//     PlcTask Outputs/GVL_iXlinker.EtherCAT_Master_BKCUCX.TcTerminals210_EK1100_2.TcTerminals210_2BK1250.A_0027_KL_6904_Safety_Logic_7_TwinSAFE_Connections.Channel_1.Safety_IB_3 <-> Channel 1/Safety IB 3
//     PlcTask Outputs/GVL_iXlinker.EtherCAT_Master_BKCUCX.TcTerminals210_EK1100_2.TcTerminals210_2BK1250.A_0027_KL_6904_Safety_Logic_7_TwinSAFE_Connections.Channel_1.Safety_IB_4 <-> Channel 1/Safety IB 4
//     PlcTask Outputs/GVL_iXlinker.EtherCAT_Master_BKCUCX.TcTerminals210_EK1100_2.TcTerminals210_2BK1250.A_0027_KL_6904_Safety_Logic_7_TwinSAFE_Connections.Channel_1.Safety_IB_5 <-> Channel 1/Safety IB 5
//     PlcTask Outputs/GVL_iXlinker.EtherCAT_Master_BKCUCX.TcTerminals210_EK1100_2.TcTerminals210_2BK1250.A_0027_KL_6904_Safety_Logic_7_TwinSAFE_Connections.Channel_1.Safety_IB_6 <-> Channel 1/Safety IB 6
//     PlcTask Outputs/GVL_iXlinker.EtherCAT_Master_BKCUCX.TcTerminals210_EK1100_2.TcTerminals210_2BK1250.A_0027_KL_6904_Safety_Logic_7_TwinSAFE_Connections.Channel_1.Safety_IB_7 <-> Channel 1/Safety IB 7
//   PLC/PLC Instance <-> EtherCAT Master BKCUCX/TcTerminals210_EK1100_2/TcTerminals210_2BK1250/A_0028(KL 6904, Safety Logic (15 TwinSAFE Connections))
//     PlcTask Inputs/GVL_iXlinker.EtherCAT_Master_BKCUCX.TcTerminals210_EK1100_2.TcTerminals210_2BK1250.A_0028_KL_6904_Safety_Logic_15_TwinSAFE_Connections.Channel_1.Status <-> Channel 1/Status
//     PlcTask Inputs/GVL_iXlinker.EtherCAT_Master_BKCUCX.TcTerminals210_EK1100_2.TcTerminals210_2BK1250.A_0028_KL_6904_Safety_Logic_15_TwinSAFE_Connections.Channel_1.Register_In <-> Channel 1/Register In
//     PlcTask Inputs/GVL_iXlinker.EtherCAT_Master_BKCUCX.TcTerminals210_EK1100_2.TcTerminals210_2BK1250.A_0028_KL_6904_Safety_Logic_15_TwinSAFE_Connections.Channel_1.Standard_QX_1 <-> Channel 1/Standard QX 1
//     PlcTask Inputs/GVL_iXlinker.EtherCAT_Master_BKCUCX.TcTerminals210_EK1100_2.TcTerminals210_2BK1250.A_0028_KL_6904_Safety_Logic_15_TwinSAFE_Connections.Channel_1.Standard_QX_2 <-> Channel 1/Standard QX 2
//     PlcTask Inputs/GVL_iXlinker.EtherCAT_Master_BKCUCX.TcTerminals210_EK1100_2.TcTerminals210_2BK1250.A_0028_KL_6904_Safety_Logic_15_TwinSAFE_Connections.Channel_1.Standard_QX_3 <-> Channel 1/Standard QX 3
//     PlcTask Inputs/GVL_iXlinker.EtherCAT_Master_BKCUCX.TcTerminals210_EK1100_2.TcTerminals210_2BK1250.A_0028_KL_6904_Safety_Logic_15_TwinSAFE_Connections.Channel_1.Safety_QB_1 <-> Channel 1/Safety QB 1
//     PlcTask Inputs/GVL_iXlinker.EtherCAT_Master_BKCUCX.TcTerminals210_EK1100_2.TcTerminals210_2BK1250.A_0028_KL_6904_Safety_Logic_15_TwinSAFE_Connections.Channel_1.Safety_QB_2 <-> Channel 1/Safety QB 2
//     PlcTask Inputs/GVL_iXlinker.EtherCAT_Master_BKCUCX.TcTerminals210_EK1100_2.TcTerminals210_2BK1250.A_0028_KL_6904_Safety_Logic_15_TwinSAFE_Connections.Channel_1.Safety_QB_3 <-> Channel 1/Safety QB 3
//     PlcTask Inputs/GVL_iXlinker.EtherCAT_Master_BKCUCX.TcTerminals210_EK1100_2.TcTerminals210_2BK1250.A_0028_KL_6904_Safety_Logic_15_TwinSAFE_Connections.Channel_1.Safety_QB_4 <-> Channel 1/Safety QB 4
//     PlcTask Inputs/GVL_iXlinker.EtherCAT_Master_BKCUCX.TcTerminals210_EK1100_2.TcTerminals210_2BK1250.A_0028_KL_6904_Safety_Logic_15_TwinSAFE_Connections.Channel_1.Safety_QB_5 <-> Channel 1/Safety QB 5
//     PlcTask Inputs/GVL_iXlinker.EtherCAT_Master_BKCUCX.TcTerminals210_EK1100_2.TcTerminals210_2BK1250.A_0028_KL_6904_Safety_Logic_15_TwinSAFE_Connections.Channel_1.Safety_QB_6 <-> Channel 1/Safety QB 6
//     PlcTask Inputs/GVL_iXlinker.EtherCAT_Master_BKCUCX.TcTerminals210_EK1100_2.TcTerminals210_2BK1250.A_0028_KL_6904_Safety_Logic_15_TwinSAFE_Connections.Channel_1.Safety_QB_7 <-> Channel 1/Safety QB 7
//     PlcTask Inputs/GVL_iXlinker.EtherCAT_Master_BKCUCX.TcTerminals210_EK1100_2.TcTerminals210_2BK1250.A_0028_KL_6904_Safety_Logic_15_TwinSAFE_Connections.Channel_1.Safety_QB_8 <-> Channel 1/Safety QB 8
//     PlcTask Inputs/GVL_iXlinker.EtherCAT_Master_BKCUCX.TcTerminals210_EK1100_2.TcTerminals210_2BK1250.A_0028_KL_6904_Safety_Logic_15_TwinSAFE_Connections.Channel_1.Safety_QB_9 <-> Channel 1/Safety QB 9
//     PlcTask Inputs/GVL_iXlinker.EtherCAT_Master_BKCUCX.TcTerminals210_EK1100_2.TcTerminals210_2BK1250.A_0028_KL_6904_Safety_Logic_15_TwinSAFE_Connections.Channel_1.Safety_QB_10 <-> Channel 1/Safety QB 10
//     PlcTask Inputs/GVL_iXlinker.EtherCAT_Master_BKCUCX.TcTerminals210_EK1100_2.TcTerminals210_2BK1250.A_0028_KL_6904_Safety_Logic_15_TwinSAFE_Connections.Channel_1.Safety_QB_11 <-> Channel 1/Safety QB 11
//     PlcTask Inputs/GVL_iXlinker.EtherCAT_Master_BKCUCX.TcTerminals210_EK1100_2.TcTerminals210_2BK1250.A_0028_KL_6904_Safety_Logic_15_TwinSAFE_Connections.Channel_1.Safety_QB_12 <-> Channel 1/Safety QB 12
//     PlcTask Inputs/GVL_iXlinker.EtherCAT_Master_BKCUCX.TcTerminals210_EK1100_2.TcTerminals210_2BK1250.A_0028_KL_6904_Safety_Logic_15_TwinSAFE_Connections.Channel_1.Safety_QB_13 <-> Channel 1/Safety QB 13
//     PlcTask Inputs/GVL_iXlinker.EtherCAT_Master_BKCUCX.TcTerminals210_EK1100_2.TcTerminals210_2BK1250.A_0028_KL_6904_Safety_Logic_15_TwinSAFE_Connections.Channel_1.Safety_QB_14 <-> Channel 1/Safety QB 14
//     PlcTask Inputs/GVL_iXlinker.EtherCAT_Master_BKCUCX.TcTerminals210_EK1100_2.TcTerminals210_2BK1250.A_0028_KL_6904_Safety_Logic_15_TwinSAFE_Connections.Channel_1.Safety_QB_15 <-> Channel 1/Safety QB 15
//     PlcTask Outputs/GVL_iXlinker.EtherCAT_Master_BKCUCX.TcTerminals210_EK1100_2.TcTerminals210_2BK1250.A_0028_KL_6904_Safety_Logic_15_TwinSAFE_Connections.Channel_1.Control <-> Channel 1/Control
//     PlcTask Outputs/GVL_iXlinker.EtherCAT_Master_BKCUCX.TcTerminals210_EK1100_2.TcTerminals210_2BK1250.A_0028_KL_6904_Safety_Logic_15_TwinSAFE_Connections.Channel_1.Register_Out <-> Channel 1/Register Out
//     PlcTask Outputs/GVL_iXlinker.EtherCAT_Master_BKCUCX.TcTerminals210_EK1100_2.TcTerminals210_2BK1250.A_0028_KL_6904_Safety_Logic_15_TwinSAFE_Connections.Channel_1.Standard_IX_1 <-> Channel 1/Standard IX 1
//     PlcTask Outputs/GVL_iXlinker.EtherCAT_Master_BKCUCX.TcTerminals210_EK1100_2.TcTerminals210_2BK1250.A_0028_KL_6904_Safety_Logic_15_TwinSAFE_Connections.Channel_1.Standard_IX_2 <-> Channel 1/Standard IX 2
//     PlcTask Outputs/GVL_iXlinker.EtherCAT_Master_BKCUCX.TcTerminals210_EK1100_2.TcTerminals210_2BK1250.A_0028_KL_6904_Safety_Logic_15_TwinSAFE_Connections.Channel_1.Standard_IX_3 <-> Channel 1/Standard IX 3
//     PlcTask Outputs/GVL_iXlinker.EtherCAT_Master_BKCUCX.TcTerminals210_EK1100_2.TcTerminals210_2BK1250.A_0028_KL_6904_Safety_Logic_15_TwinSAFE_Connections.Channel_1.Safety_IB_1 <-> Channel 1/Safety IB 1
//     PlcTask Outputs/GVL_iXlinker.EtherCAT_Master_BKCUCX.TcTerminals210_EK1100_2.TcTerminals210_2BK1250.A_0028_KL_6904_Safety_Logic_15_TwinSAFE_Connections.Channel_1.Safety_IB_2 <-> Channel 1/Safety IB 2
//     PlcTask Outputs/GVL_iXlinker.EtherCAT_Master_BKCUCX.TcTerminals210_EK1100_2.TcTerminals210_2BK1250.A_0028_KL_6904_Safety_Logic_15_TwinSAFE_Connections.Channel_1.Safety_IB_3 <-> Channel 1/Safety IB 3
//     PlcTask Outputs/GVL_iXlinker.EtherCAT_Master_BKCUCX.TcTerminals210_EK1100_2.TcTerminals210_2BK1250.A_0028_KL_6904_Safety_Logic_15_TwinSAFE_Connections.Channel_1.Safety_IB_4 <-> Channel 1/Safety IB 4
//     PlcTask Outputs/GVL_iXlinker.EtherCAT_Master_BKCUCX.TcTerminals210_EK1100_2.TcTerminals210_2BK1250.A_0028_KL_6904_Safety_Logic_15_TwinSAFE_Connections.Channel_1.Safety_IB_5 <-> Channel 1/Safety IB 5
//     PlcTask Outputs/GVL_iXlinker.EtherCAT_Master_BKCUCX.TcTerminals210_EK1100_2.TcTerminals210_2BK1250.A_0028_KL_6904_Safety_Logic_15_TwinSAFE_Connections.Channel_1.Safety_IB_6 <-> Channel 1/Safety IB 6
//     PlcTask Outputs/GVL_iXlinker.EtherCAT_Master_BKCUCX.TcTerminals210_EK1100_2.TcTerminals210_2BK1250.A_0028_KL_6904_Safety_Logic_15_TwinSAFE_Connections.Channel_1.Safety_IB_7 <-> Channel 1/Safety IB 7
//     PlcTask Outputs/GVL_iXlinker.EtherCAT_Master_BKCUCX.TcTerminals210_EK1100_2.TcTerminals210_2BK1250.A_0028_KL_6904_Safety_Logic_15_TwinSAFE_Connections.Channel_1.Safety_IB_8 <-> Channel 1/Safety IB 8
//     PlcTask Outputs/GVL_iXlinker.EtherCAT_Master_BKCUCX.TcTerminals210_EK1100_2.TcTerminals210_2BK1250.A_0028_KL_6904_Safety_Logic_15_TwinSAFE_Connections.Channel_1.Safety_IB_9 <-> Channel 1/Safety IB 9
//     PlcTask Outputs/GVL_iXlinker.EtherCAT_Master_BKCUCX.TcTerminals210_EK1100_2.TcTerminals210_2BK1250.A_0028_KL_6904_Safety_Logic_15_TwinSAFE_Connections.Channel_1.Safety_IB_10 <-> Channel 1/Safety IB 10
//     PlcTask Outputs/GVL_iXlinker.EtherCAT_Master_BKCUCX.TcTerminals210_EK1100_2.TcTerminals210_2BK1250.A_0028_KL_6904_Safety_Logic_15_TwinSAFE_Connections.Channel_1.Safety_IB_11 <-> Channel 1/Safety IB 11
//     PlcTask Outputs/GVL_iXlinker.EtherCAT_Master_BKCUCX.TcTerminals210_EK1100_2.TcTerminals210_2BK1250.A_0028_KL_6904_Safety_Logic_15_TwinSAFE_Connections.Channel_1.Safety_IB_12 <-> Channel 1/Safety IB 12
//     PlcTask Outputs/GVL_iXlinker.EtherCAT_Master_BKCUCX.TcTerminals210_EK1100_2.TcTerminals210_2BK1250.A_0028_KL_6904_Safety_Logic_15_TwinSAFE_Connections.Channel_1.Safety_IB_13 <-> Channel 1/Safety IB 13
//     PlcTask Outputs/GVL_iXlinker.EtherCAT_Master_BKCUCX.TcTerminals210_EK1100_2.TcTerminals210_2BK1250.A_0028_KL_6904_Safety_Logic_15_TwinSAFE_Connections.Channel_1.Safety_IB_14 <-> Channel 1/Safety IB 14
//     PlcTask Outputs/GVL_iXlinker.EtherCAT_Master_BKCUCX.TcTerminals210_EK1100_2.TcTerminals210_2BK1250.A_0028_KL_6904_Safety_Logic_15_TwinSAFE_Connections.Channel_1.Safety_IB_15 <-> Channel 1/Safety IB 15
//   PLC/PLC Instance <-> EtherCAT Master BKCUCX/TcTerminals210_EK1100_2/TcTerminals210_2BK1250/A_0029(KL 8001, Powerterminal (1Ch.))
//     PlcTask Inputs/GVL_iXlinker.EtherCAT_Master_BKCUCX.TcTerminals210_EK1100_2.TcTerminals210_2BK1250.A_0029_KL_8001_Powerterminal_1Ch.Channel_1.State_0 <-> Channel 1/State 0
//     PlcTask Inputs/GVL_iXlinker.EtherCAT_Master_BKCUCX.TcTerminals210_EK1100_2.TcTerminals210_2BK1250.A_0029_KL_8001_Powerterminal_1Ch.Channel_1.Data_In_0 <-> Channel 1/Data In 0
//     PlcTask Inputs/GVL_iXlinker.EtherCAT_Master_BKCUCX.TcTerminals210_EK1100_2.TcTerminals210_2BK1250.A_0029_KL_8001_Powerterminal_1Ch.Channel_1.State_Ext <-> Channel 1/State Ext.
//     PlcTask Outputs/GVL_iXlinker.EtherCAT_Master_BKCUCX.TcTerminals210_EK1100_2.TcTerminals210_2BK1250.A_0029_KL_8001_Powerterminal_1Ch.Channel_1.Ctrl_0 <-> Channel 1/Ctrl 0
//     PlcTask Outputs/GVL_iXlinker.EtherCAT_Master_BKCUCX.TcTerminals210_EK1100_2.TcTerminals210_2BK1250.A_0029_KL_8001_Powerterminal_1Ch.Channel_1.Data_Out_0 <-> Channel 1/Data Out 0
//     PlcTask Outputs/GVL_iXlinker.EtherCAT_Master_BKCUCX.TcTerminals210_EK1100_2.TcTerminals210_2BK1250.A_0029_KL_8001_Powerterminal_1Ch.Channel_1.Ctrl_Ext <-> Channel 1/Ctrl Ext.
//   PLC/PLC Instance <-> EtherCAT Master BKCUCX/TcTerminals210_EK1100_2/TcTerminals210_2BK1250/A_0030(KL 8001, Powerterminal (3 Ch.))
//     PlcTask Inputs/GVL_iXlinker.EtherCAT_Master_BKCUCX.TcTerminals210_EK1100_2.TcTerminals210_2BK1250.A_0030_KL_8001_Powerterminal_3_Ch.Channel_1.State_0 <-> Channel 1/State 0
//     PlcTask Inputs/GVL_iXlinker.EtherCAT_Master_BKCUCX.TcTerminals210_EK1100_2.TcTerminals210_2BK1250.A_0030_KL_8001_Powerterminal_3_Ch.Channel_1.State_1 <-> Channel 1/State 1
//     PlcTask Inputs/GVL_iXlinker.EtherCAT_Master_BKCUCX.TcTerminals210_EK1100_2.TcTerminals210_2BK1250.A_0030_KL_8001_Powerterminal_3_Ch.Channel_1.State_2 <-> Channel 1/State 2
//     PlcTask Inputs/GVL_iXlinker.EtherCAT_Master_BKCUCX.TcTerminals210_EK1100_2.TcTerminals210_2BK1250.A_0030_KL_8001_Powerterminal_3_Ch.Channel_1.Data_In_0 <-> Channel 1/Data In 0
//     PlcTask Inputs/GVL_iXlinker.EtherCAT_Master_BKCUCX.TcTerminals210_EK1100_2.TcTerminals210_2BK1250.A_0030_KL_8001_Powerterminal_3_Ch.Channel_1.Data_In_1 <-> Channel 1/Data In 1
//     PlcTask Inputs/GVL_iXlinker.EtherCAT_Master_BKCUCX.TcTerminals210_EK1100_2.TcTerminals210_2BK1250.A_0030_KL_8001_Powerterminal_3_Ch.Channel_1.Data_In_2 <-> Channel 1/Data In 2
//     PlcTask Inputs/GVL_iXlinker.EtherCAT_Master_BKCUCX.TcTerminals210_EK1100_2.TcTerminals210_2BK1250.A_0030_KL_8001_Powerterminal_3_Ch.Channel_1.State_Ext <-> Channel 1/State Ext.
//     PlcTask Outputs/GVL_iXlinker.EtherCAT_Master_BKCUCX.TcTerminals210_EK1100_2.TcTerminals210_2BK1250.A_0030_KL_8001_Powerterminal_3_Ch.Channel_1.Ctrl_0 <-> Channel 1/Ctrl 0
//     PlcTask Outputs/GVL_iXlinker.EtherCAT_Master_BKCUCX.TcTerminals210_EK1100_2.TcTerminals210_2BK1250.A_0030_KL_8001_Powerterminal_3_Ch.Channel_1.Ctrl_1 <-> Channel 1/Ctrl 1
//     PlcTask Outputs/GVL_iXlinker.EtherCAT_Master_BKCUCX.TcTerminals210_EK1100_2.TcTerminals210_2BK1250.A_0030_KL_8001_Powerterminal_3_Ch.Channel_1.Ctrl_2 <-> Channel 1/Ctrl 2
//     PlcTask Outputs/GVL_iXlinker.EtherCAT_Master_BKCUCX.TcTerminals210_EK1100_2.TcTerminals210_2BK1250.A_0030_KL_8001_Powerterminal_3_Ch.Channel_1.Data_Out_0 <-> Channel 1/Data Out 0
//     PlcTask Outputs/GVL_iXlinker.EtherCAT_Master_BKCUCX.TcTerminals210_EK1100_2.TcTerminals210_2BK1250.A_0030_KL_8001_Powerterminal_3_Ch.Channel_1.Data_Out_1 <-> Channel 1/Data Out 1
//     PlcTask Outputs/GVL_iXlinker.EtherCAT_Master_BKCUCX.TcTerminals210_EK1100_2.TcTerminals210_2BK1250.A_0030_KL_8001_Powerterminal_3_Ch.Channel_1.Data_Out_2 <-> Channel 1/Data Out 2
//     PlcTask Outputs/GVL_iXlinker.EtherCAT_Master_BKCUCX.TcTerminals210_EK1100_2.TcTerminals210_2BK1250.A_0030_KL_8001_Powerterminal_3_Ch.Channel_1.Ctrl_Ext <-> Channel 1/Ctrl Ext.
//   PLC/PLC Instance <-> EtherCAT Master BKCUCX/TcTerminals210_EK1100_2/TcTerminals210_2BK1250/A_0031(KL 8519, 16 digital Input)
//     PlcTask Inputs/GVL_iXlinker.EtherCAT_Master_BKCUCX.TcTerminals210_EK1100_2.TcTerminals210_2BK1250.A_0031_KL_8519_16_digital_Input.Channel_1.State <-> Channel 1/State
//     PlcTask Inputs/GVL_iXlinker.EtherCAT_Master_BKCUCX.TcTerminals210_EK1100_2.TcTerminals210_2BK1250.A_0031_KL_8519_16_digital_Input.Channel_1.Data_In_1 <-> Channel 1/Data In 1
//     PlcTask Inputs/GVL_iXlinker.EtherCAT_Master_BKCUCX.TcTerminals210_EK1100_2.TcTerminals210_2BK1250.A_0031_KL_8519_16_digital_Input.Channel_1.Data_In_2 <-> Channel 1/Data In 2
//     PlcTask Outputs/GVL_iXlinker.EtherCAT_Master_BKCUCX.TcTerminals210_EK1100_2.TcTerminals210_2BK1250.A_0031_KL_8519_16_digital_Input.Channel_1.Ctrl <-> Channel 1/Ctrl
//     PlcTask Outputs/GVL_iXlinker.EtherCAT_Master_BKCUCX.TcTerminals210_EK1100_2.TcTerminals210_2BK1250.A_0031_KL_8519_16_digital_Input.Channel_1.LED_Out_green_1 <-> Channel 1/LED Out green 1
//     PlcTask Outputs/GVL_iXlinker.EtherCAT_Master_BKCUCX.TcTerminals210_EK1100_2.TcTerminals210_2BK1250.A_0031_KL_8519_16_digital_Input.Channel_1.LED_Out_green_2 <-> Channel 1/LED Out green 2
//     PlcTask Outputs/GVL_iXlinker.EtherCAT_Master_BKCUCX.TcTerminals210_EK1100_2.TcTerminals210_2BK1250.A_0031_KL_8519_16_digital_Input.Channel_1.LED_Out_red_1 <-> Channel 1/LED Out red 1
//     PlcTask Outputs/GVL_iXlinker.EtherCAT_Master_BKCUCX.TcTerminals210_EK1100_2.TcTerminals210_2BK1250.A_0031_KL_8519_16_digital_Input.Channel_1.LED_Out_red_2 <-> Channel 1/LED Out red 2
//   PLC/PLC Instance <-> EtherCAT Master BKCUCX/TcTerminals210_EK1100_2/TcTerminals210_2BK1250/A_0032(KL 8524, 2x4 digital Output)
//     PlcTask Inputs/GVL_iXlinker.EtherCAT_Master_BKCUCX.TcTerminals210_EK1100_2.TcTerminals210_2BK1250.A_0032_KL_8524_2x4_digital_Output.Channel_1.State <-> Channel 1/State
//     PlcTask Inputs/GVL_iXlinker.EtherCAT_Master_BKCUCX.TcTerminals210_EK1100_2.TcTerminals210_2BK1250.A_0032_KL_8524_2x4_digital_Output.Channel_1.Auto_Manual_Channel <-> Channel 1/Auto/Manual Channel
//     PlcTask Inputs/GVL_iXlinker.EtherCAT_Master_BKCUCX.TcTerminals210_EK1100_2.TcTerminals210_2BK1250.A_0032_KL_8524_2x4_digital_Output.Channel_1.Switch_mode <-> Channel 1/Switch mode
//     PlcTask Inputs/GVL_iXlinker.EtherCAT_Master_BKCUCX.TcTerminals210_EK1100_2.TcTerminals210_2BK1250.A_0032_KL_8524_2x4_digital_Output.Channel_1.On_Off_Channel <-> Channel 1/On/Off Channel
//     PlcTask Outputs/GVL_iXlinker.EtherCAT_Master_BKCUCX.TcTerminals210_EK1100_2.TcTerminals210_2BK1250.A_0032_KL_8524_2x4_digital_Output.Channel_1.Ctrl <-> Channel 1/Ctrl
//     PlcTask Outputs/GVL_iXlinker.EtherCAT_Master_BKCUCX.TcTerminals210_EK1100_2.TcTerminals210_2BK1250.A_0032_KL_8524_2x4_digital_Output.Channel_1.Switch_mode_Out <-> Channel 1/Switch mode Out
//     PlcTask Outputs/GVL_iXlinker.EtherCAT_Master_BKCUCX.TcTerminals210_EK1100_2.TcTerminals210_2BK1250.A_0032_KL_8524_2x4_digital_Output.Channel_1.Data_Reg_Com <-> Channel 1/Data (Reg.Com)
//     PlcTask Outputs/GVL_iXlinker.EtherCAT_Master_BKCUCX.TcTerminals210_EK1100_2.TcTerminals210_2BK1250.A_0032_KL_8524_2x4_digital_Output.Channel_1.LED_Out_green <-> Channel 1/LED Out green
//     PlcTask Outputs/GVL_iXlinker.EtherCAT_Master_BKCUCX.TcTerminals210_EK1100_2.TcTerminals210_2BK1250.A_0032_KL_8524_2x4_digital_Output.Channel_1.LED_Out_yellow <-> Channel 1/LED Out yellow
//   PLC/PLC Instance <-> EtherCAT Master BKCUCX/TcTerminals210_EK1100_2/TcTerminals210_2BK1250/A_0033(KL 8528, 8 digital Output)
//     PlcTask Inputs/GVL_iXlinker.EtherCAT_Master_BKCUCX.TcTerminals210_EK1100_2.TcTerminals210_2BK1250.A_0033_KL_8528_8_digital_Output.Channel_1.State <-> Channel 1/State
//     PlcTask Inputs/GVL_iXlinker.EtherCAT_Master_BKCUCX.TcTerminals210_EK1100_2.TcTerminals210_2BK1250.A_0033_KL_8528_8_digital_Output.Channel_1.Auto_Manual_Channel <-> Channel 1/Auto/Manual Channel
//     PlcTask Inputs/GVL_iXlinker.EtherCAT_Master_BKCUCX.TcTerminals210_EK1100_2.TcTerminals210_2BK1250.A_0033_KL_8528_8_digital_Output.Channel_1.On_Off_Channel <-> Channel 1/On/Off Channel
//     PlcTask Outputs/GVL_iXlinker.EtherCAT_Master_BKCUCX.TcTerminals210_EK1100_2.TcTerminals210_2BK1250.A_0033_KL_8528_8_digital_Output.Channel_1.Ctrl <-> Channel 1/Ctrl
//     PlcTask Outputs/GVL_iXlinker.EtherCAT_Master_BKCUCX.TcTerminals210_EK1100_2.TcTerminals210_2BK1250.A_0033_KL_8528_8_digital_Output.Channel_1.Out <-> Channel 1/Out
//     PlcTask Outputs/GVL_iXlinker.EtherCAT_Master_BKCUCX.TcTerminals210_EK1100_2.TcTerminals210_2BK1250.A_0033_KL_8528_8_digital_Output.Channel_1.Data_Reg_Com <-> Channel 1/Data (Reg.Com)
//     PlcTask Outputs/GVL_iXlinker.EtherCAT_Master_BKCUCX.TcTerminals210_EK1100_2.TcTerminals210_2BK1250.A_0033_KL_8528_8_digital_Output.Channel_1.LED_Out_green <-> Channel 1/LED Out green
//     PlcTask Outputs/GVL_iXlinker.EtherCAT_Master_BKCUCX.TcTerminals210_EK1100_2.TcTerminals210_2BK1250.A_0033_KL_8528_8_digital_Output.Channel_1.LED_Out_yellow <-> Channel 1/LED Out yellow
//   PLC/PLC Instance <-> EtherCAT Master BKCUCX/TcTerminals210_EK1100_2/TcTerminals210_2BK1250/A_0034(KL 8548, 8 Ch. ana. Output (0..10V))
//     PlcTask Inputs/GVL_iXlinker.EtherCAT_Master_BKCUCX.TcTerminals210_EK1100_2.TcTerminals210_2BK1250.A_0034_KL_8548_8_Ch_ana_Output_0_10V.Channel_1.State <-> Channel 1/State
//     PlcTask Inputs/GVL_iXlinker.EtherCAT_Master_BKCUCX.TcTerminals210_EK1100_2.TcTerminals210_2BK1250.A_0034_KL_8548_8_Ch_ana_Output_0_10V.Channel_2.State <-> Channel 2/State
//     PlcTask Inputs/GVL_iXlinker.EtherCAT_Master_BKCUCX.TcTerminals210_EK1100_2.TcTerminals210_2BK1250.A_0034_KL_8548_8_Ch_ana_Output_0_10V.Channel_3.State <-> Channel 3/State
//     PlcTask Inputs/GVL_iXlinker.EtherCAT_Master_BKCUCX.TcTerminals210_EK1100_2.TcTerminals210_2BK1250.A_0034_KL_8548_8_Ch_ana_Output_0_10V.Channel_4.State <-> Channel 4/State
//     PlcTask Inputs/GVL_iXlinker.EtherCAT_Master_BKCUCX.TcTerminals210_EK1100_2.TcTerminals210_2BK1250.A_0034_KL_8548_8_Ch_ana_Output_0_10V.Channel_5.State <-> Channel 5/State
//     PlcTask Inputs/GVL_iXlinker.EtherCAT_Master_BKCUCX.TcTerminals210_EK1100_2.TcTerminals210_2BK1250.A_0034_KL_8548_8_Ch_ana_Output_0_10V.Channel_6.State <-> Channel 6/State
//     PlcTask Inputs/GVL_iXlinker.EtherCAT_Master_BKCUCX.TcTerminals210_EK1100_2.TcTerminals210_2BK1250.A_0034_KL_8548_8_Ch_ana_Output_0_10V.Channel_7.State <-> Channel 7/State
//     PlcTask Inputs/GVL_iXlinker.EtherCAT_Master_BKCUCX.TcTerminals210_EK1100_2.TcTerminals210_2BK1250.A_0034_KL_8548_8_Ch_ana_Output_0_10V.Channel_8.State <-> Channel 8/State
//     PlcTask Inputs/GVL_iXlinker.EtherCAT_Master_BKCUCX.TcTerminals210_EK1100_2.TcTerminals210_2BK1250.A_0034_KL_8548_8_Ch_ana_Output_0_10V.Channel_1.Data_In <-> Channel 1/Data In
//     PlcTask Inputs/GVL_iXlinker.EtherCAT_Master_BKCUCX.TcTerminals210_EK1100_2.TcTerminals210_2BK1250.A_0034_KL_8548_8_Ch_ana_Output_0_10V.Channel_2.Data_In <-> Channel 2/Data In
//     PlcTask Inputs/GVL_iXlinker.EtherCAT_Master_BKCUCX.TcTerminals210_EK1100_2.TcTerminals210_2BK1250.A_0034_KL_8548_8_Ch_ana_Output_0_10V.Channel_3.Data_In <-> Channel 3/Data In
//     PlcTask Inputs/GVL_iXlinker.EtherCAT_Master_BKCUCX.TcTerminals210_EK1100_2.TcTerminals210_2BK1250.A_0034_KL_8548_8_Ch_ana_Output_0_10V.Channel_4.Data_In <-> Channel 4/Data In
//     PlcTask Inputs/GVL_iXlinker.EtherCAT_Master_BKCUCX.TcTerminals210_EK1100_2.TcTerminals210_2BK1250.A_0034_KL_8548_8_Ch_ana_Output_0_10V.Channel_5.Data_In <-> Channel 5/Data In
//     PlcTask Inputs/GVL_iXlinker.EtherCAT_Master_BKCUCX.TcTerminals210_EK1100_2.TcTerminals210_2BK1250.A_0034_KL_8548_8_Ch_ana_Output_0_10V.Channel_6.Data_In <-> Channel 6/Data In
//     PlcTask Inputs/GVL_iXlinker.EtherCAT_Master_BKCUCX.TcTerminals210_EK1100_2.TcTerminals210_2BK1250.A_0034_KL_8548_8_Ch_ana_Output_0_10V.Channel_7.Data_In <-> Channel 7/Data In
//     PlcTask Inputs/GVL_iXlinker.EtherCAT_Master_BKCUCX.TcTerminals210_EK1100_2.TcTerminals210_2BK1250.A_0034_KL_8548_8_Ch_ana_Output_0_10V.Channel_8.Data_In <-> Channel 8/Data In
//     PlcTask Outputs/GVL_iXlinker.EtherCAT_Master_BKCUCX.TcTerminals210_EK1100_2.TcTerminals210_2BK1250.A_0034_KL_8548_8_Ch_ana_Output_0_10V.Channel_1.Ctrl <-> Channel 1/Ctrl
//     PlcTask Outputs/GVL_iXlinker.EtherCAT_Master_BKCUCX.TcTerminals210_EK1100_2.TcTerminals210_2BK1250.A_0034_KL_8548_8_Ch_ana_Output_0_10V.Channel_2.Ctrl <-> Channel 2/Ctrl
//     PlcTask Outputs/GVL_iXlinker.EtherCAT_Master_BKCUCX.TcTerminals210_EK1100_2.TcTerminals210_2BK1250.A_0034_KL_8548_8_Ch_ana_Output_0_10V.Channel_3.Ctrl <-> Channel 3/Ctrl
//     PlcTask Outputs/GVL_iXlinker.EtherCAT_Master_BKCUCX.TcTerminals210_EK1100_2.TcTerminals210_2BK1250.A_0034_KL_8548_8_Ch_ana_Output_0_10V.Channel_4.Ctrl <-> Channel 4/Ctrl
//     PlcTask Outputs/GVL_iXlinker.EtherCAT_Master_BKCUCX.TcTerminals210_EK1100_2.TcTerminals210_2BK1250.A_0034_KL_8548_8_Ch_ana_Output_0_10V.Channel_5.Ctrl <-> Channel 5/Ctrl
//     PlcTask Outputs/GVL_iXlinker.EtherCAT_Master_BKCUCX.TcTerminals210_EK1100_2.TcTerminals210_2BK1250.A_0034_KL_8548_8_Ch_ana_Output_0_10V.Channel_6.Ctrl <-> Channel 6/Ctrl
//     PlcTask Outputs/GVL_iXlinker.EtherCAT_Master_BKCUCX.TcTerminals210_EK1100_2.TcTerminals210_2BK1250.A_0034_KL_8548_8_Ch_ana_Output_0_10V.Channel_7.Ctrl <-> Channel 7/Ctrl
//     PlcTask Outputs/GVL_iXlinker.EtherCAT_Master_BKCUCX.TcTerminals210_EK1100_2.TcTerminals210_2BK1250.A_0034_KL_8548_8_Ch_ana_Output_0_10V.Channel_8.Ctrl <-> Channel 8/Ctrl
//     PlcTask Outputs/GVL_iXlinker.EtherCAT_Master_BKCUCX.TcTerminals210_EK1100_2.TcTerminals210_2BK1250.A_0034_KL_8548_8_Ch_ana_Output_0_10V.Channel_1.Data_Out <-> Channel 1/Data Out
//     PlcTask Outputs/GVL_iXlinker.EtherCAT_Master_BKCUCX.TcTerminals210_EK1100_2.TcTerminals210_2BK1250.A_0034_KL_8548_8_Ch_ana_Output_0_10V.Channel_2.Data_Out <-> Channel 2/Data Out
//     PlcTask Outputs/GVL_iXlinker.EtherCAT_Master_BKCUCX.TcTerminals210_EK1100_2.TcTerminals210_2BK1250.A_0034_KL_8548_8_Ch_ana_Output_0_10V.Channel_3.Data_Out <-> Channel 3/Data Out
//     PlcTask Outputs/GVL_iXlinker.EtherCAT_Master_BKCUCX.TcTerminals210_EK1100_2.TcTerminals210_2BK1250.A_0034_KL_8548_8_Ch_ana_Output_0_10V.Channel_4.Data_Out <-> Channel 4/Data Out
//     PlcTask Outputs/GVL_iXlinker.EtherCAT_Master_BKCUCX.TcTerminals210_EK1100_2.TcTerminals210_2BK1250.A_0034_KL_8548_8_Ch_ana_Output_0_10V.Channel_5.Data_Out <-> Channel 5/Data Out
//     PlcTask Outputs/GVL_iXlinker.EtherCAT_Master_BKCUCX.TcTerminals210_EK1100_2.TcTerminals210_2BK1250.A_0034_KL_8548_8_Ch_ana_Output_0_10V.Channel_6.Data_Out <-> Channel 6/Data Out
//     PlcTask Outputs/GVL_iXlinker.EtherCAT_Master_BKCUCX.TcTerminals210_EK1100_2.TcTerminals210_2BK1250.A_0034_KL_8548_8_Ch_ana_Output_0_10V.Channel_7.Data_Out <-> Channel 7/Data Out
//     PlcTask Outputs/GVL_iXlinker.EtherCAT_Master_BKCUCX.TcTerminals210_EK1100_2.TcTerminals210_2BK1250.A_0034_KL_8548_8_Ch_ana_Output_0_10V.Channel_8.Data_Out <-> Channel 8/Data Out
//   PLC/PLC Instance <-> EtherCAT Master BKCUCX/TcTerminals210_EK1100_2/TcTerminals210_2BK1250/A_0035(KL 8610, 1 Ch. Adapter KL8601)
//     PlcTask Inputs/GVL_iXlinker.EtherCAT_Master_BKCUCX.TcTerminals210_EK1100_2.TcTerminals210_2BK1250.A_0035_KL_8610_1_Ch_Adapter_KL8601.KL8601_1.State <-> KL8601 - 1/State
//     PlcTask Inputs/GVL_iXlinker.EtherCAT_Master_BKCUCX.TcTerminals210_EK1100_2.TcTerminals210_2BK1250.A_0035_KL_8610_1_Ch_Adapter_KL8601.KL8601_1.Data_In <-> KL8601 - 1/Data In
//     PlcTask Outputs/GVL_iXlinker.EtherCAT_Master_BKCUCX.TcTerminals210_EK1100_2.TcTerminals210_2BK1250.A_0035_KL_8610_1_Ch_Adapter_KL8601.KL8601_1.Ctrl <-> KL8601 - 1/Ctrl
//     PlcTask Outputs/GVL_iXlinker.EtherCAT_Master_BKCUCX.TcTerminals210_EK1100_2.TcTerminals210_2BK1250.A_0035_KL_8610_1_Ch_Adapter_KL8601.KL8601_1.Data_Out <-> KL8601 - 1/Data Out
//   PLC/PLC Instance <-> EtherCAT Master BKCUCX/TcTerminals210_EK1100_2/TcTerminals210_2BK1250/A_0036(KL 8610, 2 Ch. Adapter KL8601)
//     PlcTask Inputs/GVL_iXlinker.EtherCAT_Master_BKCUCX.TcTerminals210_EK1100_2.TcTerminals210_2BK1250.A_0036_KL_8610_2_Ch_Adapter_KL8601.KL8601_1.State <-> KL8601 - 1/State
//     PlcTask Inputs/GVL_iXlinker.EtherCAT_Master_BKCUCX.TcTerminals210_EK1100_2.TcTerminals210_2BK1250.A_0036_KL_8610_2_Ch_Adapter_KL8601.KL8601_2.State <-> KL8601 - 2/State
//     PlcTask Inputs/GVL_iXlinker.EtherCAT_Master_BKCUCX.TcTerminals210_EK1100_2.TcTerminals210_2BK1250.A_0036_KL_8610_2_Ch_Adapter_KL8601.KL8601_1.Data_In <-> KL8601 - 1/Data In
//     PlcTask Inputs/GVL_iXlinker.EtherCAT_Master_BKCUCX.TcTerminals210_EK1100_2.TcTerminals210_2BK1250.A_0036_KL_8610_2_Ch_Adapter_KL8601.KL8601_2.Data_In <-> KL8601 - 2/Data In
//     PlcTask Outputs/GVL_iXlinker.EtherCAT_Master_BKCUCX.TcTerminals210_EK1100_2.TcTerminals210_2BK1250.A_0036_KL_8610_2_Ch_Adapter_KL8601.KL8601_1.Ctrl <-> KL8601 - 1/Ctrl
//     PlcTask Outputs/GVL_iXlinker.EtherCAT_Master_BKCUCX.TcTerminals210_EK1100_2.TcTerminals210_2BK1250.A_0036_KL_8610_2_Ch_Adapter_KL8601.KL8601_2.Ctrl <-> KL8601 - 2/Ctrl
//     PlcTask Outputs/GVL_iXlinker.EtherCAT_Master_BKCUCX.TcTerminals210_EK1100_2.TcTerminals210_2BK1250.A_0036_KL_8610_2_Ch_Adapter_KL8601.KL8601_1.Data_Out <-> KL8601 - 1/Data Out
//     PlcTask Outputs/GVL_iXlinker.EtherCAT_Master_BKCUCX.TcTerminals210_EK1100_2.TcTerminals210_2BK1250.A_0036_KL_8610_2_Ch_Adapter_KL8601.KL8601_2.Data_Out <-> KL8601 - 2/Data Out
//   PLC/PLC Instance <-> EtherCAT Master BKCUCX/TcTerminals210_EK1100_2/TcTerminals210_2BK1250/A_0037(KL 8610, 3 Ch. Adapter KL8601)
//     PlcTask Inputs/GVL_iXlinker.EtherCAT_Master_BKCUCX.TcTerminals210_EK1100_2.TcTerminals210_2BK1250.A_0037_KL_8610_3_Ch_Adapter_KL8601.KL8601_1.State <-> KL8601 - 1/State
//     PlcTask Inputs/GVL_iXlinker.EtherCAT_Master_BKCUCX.TcTerminals210_EK1100_2.TcTerminals210_2BK1250.A_0037_KL_8610_3_Ch_Adapter_KL8601.KL8601_2.State <-> KL8601 - 2/State
//     PlcTask Inputs/GVL_iXlinker.EtherCAT_Master_BKCUCX.TcTerminals210_EK1100_2.TcTerminals210_2BK1250.A_0037_KL_8610_3_Ch_Adapter_KL8601.KL8601_3.State <-> KL8601 - 3/State
//     PlcTask Inputs/GVL_iXlinker.EtherCAT_Master_BKCUCX.TcTerminals210_EK1100_2.TcTerminals210_2BK1250.A_0037_KL_8610_3_Ch_Adapter_KL8601.KL8601_1.Data_In <-> KL8601 - 1/Data In
//     PlcTask Inputs/GVL_iXlinker.EtherCAT_Master_BKCUCX.TcTerminals210_EK1100_2.TcTerminals210_2BK1250.A_0037_KL_8610_3_Ch_Adapter_KL8601.KL8601_2.Data_In <-> KL8601 - 2/Data In
//     PlcTask Inputs/GVL_iXlinker.EtherCAT_Master_BKCUCX.TcTerminals210_EK1100_2.TcTerminals210_2BK1250.A_0037_KL_8610_3_Ch_Adapter_KL8601.KL8601_3.Data_In <-> KL8601 - 3/Data In
//     PlcTask Outputs/GVL_iXlinker.EtherCAT_Master_BKCUCX.TcTerminals210_EK1100_2.TcTerminals210_2BK1250.A_0037_KL_8610_3_Ch_Adapter_KL8601.KL8601_1.Ctrl <-> KL8601 - 1/Ctrl
//     PlcTask Outputs/GVL_iXlinker.EtherCAT_Master_BKCUCX.TcTerminals210_EK1100_2.TcTerminals210_2BK1250.A_0037_KL_8610_3_Ch_Adapter_KL8601.KL8601_2.Ctrl <-> KL8601 - 2/Ctrl
//     PlcTask Outputs/GVL_iXlinker.EtherCAT_Master_BKCUCX.TcTerminals210_EK1100_2.TcTerminals210_2BK1250.A_0037_KL_8610_3_Ch_Adapter_KL8601.KL8601_3.Ctrl <-> KL8601 - 3/Ctrl
//     PlcTask Outputs/GVL_iXlinker.EtherCAT_Master_BKCUCX.TcTerminals210_EK1100_2.TcTerminals210_2BK1250.A_0037_KL_8610_3_Ch_Adapter_KL8601.KL8601_1.Data_Out <-> KL8601 - 1/Data Out
//     PlcTask Outputs/GVL_iXlinker.EtherCAT_Master_BKCUCX.TcTerminals210_EK1100_2.TcTerminals210_2BK1250.A_0037_KL_8610_3_Ch_Adapter_KL8601.KL8601_2.Data_Out <-> KL8601 - 2/Data Out
//     PlcTask Outputs/GVL_iXlinker.EtherCAT_Master_BKCUCX.TcTerminals210_EK1100_2.TcTerminals210_2BK1250.A_0037_KL_8610_3_Ch_Adapter_KL8601.KL8601_3.Data_Out <-> KL8601 - 3/Data Out
//   PLC/PLC Instance <-> EtherCAT Master BKCUCX/TcTerminals210_EK1100_2/TcTerminals210_2BK1250/A_0038(KL 8610, 4 Ch. Adapter KL8601)
//     PlcTask Inputs/GVL_iXlinker.EtherCAT_Master_BKCUCX.TcTerminals210_EK1100_2.TcTerminals210_2BK1250.A_0038_KL_8610_4_Ch_Adapter_KL8601.KL8601_1.State <-> KL8601 - 1/State
//     PlcTask Inputs/GVL_iXlinker.EtherCAT_Master_BKCUCX.TcTerminals210_EK1100_2.TcTerminals210_2BK1250.A_0038_KL_8610_4_Ch_Adapter_KL8601.KL8601_2.State <-> KL8601 - 2/State
//     PlcTask Inputs/GVL_iXlinker.EtherCAT_Master_BKCUCX.TcTerminals210_EK1100_2.TcTerminals210_2BK1250.A_0038_KL_8610_4_Ch_Adapter_KL8601.KL8601_3.State <-> KL8601 - 3/State
//     PlcTask Inputs/GVL_iXlinker.EtherCAT_Master_BKCUCX.TcTerminals210_EK1100_2.TcTerminals210_2BK1250.A_0038_KL_8610_4_Ch_Adapter_KL8601.KL8601_4.State <-> KL8601 - 4/State
//     PlcTask Inputs/GVL_iXlinker.EtherCAT_Master_BKCUCX.TcTerminals210_EK1100_2.TcTerminals210_2BK1250.A_0038_KL_8610_4_Ch_Adapter_KL8601.KL8601_1.Data_In <-> KL8601 - 1/Data In
//     PlcTask Inputs/GVL_iXlinker.EtherCAT_Master_BKCUCX.TcTerminals210_EK1100_2.TcTerminals210_2BK1250.A_0038_KL_8610_4_Ch_Adapter_KL8601.KL8601_2.Data_In <-> KL8601 - 2/Data In
//     PlcTask Inputs/GVL_iXlinker.EtherCAT_Master_BKCUCX.TcTerminals210_EK1100_2.TcTerminals210_2BK1250.A_0038_KL_8610_4_Ch_Adapter_KL8601.KL8601_3.Data_In <-> KL8601 - 3/Data In
//     PlcTask Inputs/GVL_iXlinker.EtherCAT_Master_BKCUCX.TcTerminals210_EK1100_2.TcTerminals210_2BK1250.A_0038_KL_8610_4_Ch_Adapter_KL8601.KL8601_4.Data_In <-> KL8601 - 4/Data In
//     PlcTask Outputs/GVL_iXlinker.EtherCAT_Master_BKCUCX.TcTerminals210_EK1100_2.TcTerminals210_2BK1250.A_0038_KL_8610_4_Ch_Adapter_KL8601.KL8601_1.Ctrl <-> KL8601 - 1/Ctrl
//     PlcTask Outputs/GVL_iXlinker.EtherCAT_Master_BKCUCX.TcTerminals210_EK1100_2.TcTerminals210_2BK1250.A_0038_KL_8610_4_Ch_Adapter_KL8601.KL8601_2.Ctrl <-> KL8601 - 2/Ctrl
//     PlcTask Outputs/GVL_iXlinker.EtherCAT_Master_BKCUCX.TcTerminals210_EK1100_2.TcTerminals210_2BK1250.A_0038_KL_8610_4_Ch_Adapter_KL8601.KL8601_3.Ctrl <-> KL8601 - 3/Ctrl
//     PlcTask Outputs/GVL_iXlinker.EtherCAT_Master_BKCUCX.TcTerminals210_EK1100_2.TcTerminals210_2BK1250.A_0038_KL_8610_4_Ch_Adapter_KL8601.KL8601_4.Ctrl <-> KL8601 - 4/Ctrl
//     PlcTask Outputs/GVL_iXlinker.EtherCAT_Master_BKCUCX.TcTerminals210_EK1100_2.TcTerminals210_2BK1250.A_0038_KL_8610_4_Ch_Adapter_KL8601.KL8601_1.Data_Out <-> KL8601 - 1/Data Out
//     PlcTask Outputs/GVL_iXlinker.EtherCAT_Master_BKCUCX.TcTerminals210_EK1100_2.TcTerminals210_2BK1250.A_0038_KL_8610_4_Ch_Adapter_KL8601.KL8601_2.Data_Out <-> KL8601 - 2/Data Out
//     PlcTask Outputs/GVL_iXlinker.EtherCAT_Master_BKCUCX.TcTerminals210_EK1100_2.TcTerminals210_2BK1250.A_0038_KL_8610_4_Ch_Adapter_KL8601.KL8601_3.Data_Out <-> KL8601 - 3/Data Out
//     PlcTask Outputs/GVL_iXlinker.EtherCAT_Master_BKCUCX.TcTerminals210_EK1100_2.TcTerminals210_2BK1250.A_0038_KL_8610_4_Ch_Adapter_KL8601.KL8601_4.Data_Out <-> KL8601 - 4/Data Out
//   PLC/PLC Instance <-> EtherCAT Master BKCUCX/TcTerminals210_EK1100_2/TcTerminals210_2BK1250/A_0039(KL 8610, 5 Ch. Adapter KL8601)
//     PlcTask Inputs/GVL_iXlinker.EtherCAT_Master_BKCUCX.TcTerminals210_EK1100_2.TcTerminals210_2BK1250.A_0039_KL_8610_5_Ch_Adapter_KL8601.KL8601_1.State <-> KL8601 - 1/State
//     PlcTask Inputs/GVL_iXlinker.EtherCAT_Master_BKCUCX.TcTerminals210_EK1100_2.TcTerminals210_2BK1250.A_0039_KL_8610_5_Ch_Adapter_KL8601.KL8601_2.State <-> KL8601 - 2/State
//     PlcTask Inputs/GVL_iXlinker.EtherCAT_Master_BKCUCX.TcTerminals210_EK1100_2.TcTerminals210_2BK1250.A_0039_KL_8610_5_Ch_Adapter_KL8601.KL8601_3.State <-> KL8601 - 3/State
//     PlcTask Inputs/GVL_iXlinker.EtherCAT_Master_BKCUCX.TcTerminals210_EK1100_2.TcTerminals210_2BK1250.A_0039_KL_8610_5_Ch_Adapter_KL8601.KL8601_4.State <-> KL8601 - 4/State
//     PlcTask Inputs/GVL_iXlinker.EtherCAT_Master_BKCUCX.TcTerminals210_EK1100_2.TcTerminals210_2BK1250.A_0039_KL_8610_5_Ch_Adapter_KL8601.KL8601_5.State <-> KL8601 - 5/State
//     PlcTask Inputs/GVL_iXlinker.EtherCAT_Master_BKCUCX.TcTerminals210_EK1100_2.TcTerminals210_2BK1250.A_0039_KL_8610_5_Ch_Adapter_KL8601.KL8601_1.Data_In <-> KL8601 - 1/Data In
//     PlcTask Inputs/GVL_iXlinker.EtherCAT_Master_BKCUCX.TcTerminals210_EK1100_2.TcTerminals210_2BK1250.A_0039_KL_8610_5_Ch_Adapter_KL8601.KL8601_2.Data_In <-> KL8601 - 2/Data In
//     PlcTask Inputs/GVL_iXlinker.EtherCAT_Master_BKCUCX.TcTerminals210_EK1100_2.TcTerminals210_2BK1250.A_0039_KL_8610_5_Ch_Adapter_KL8601.KL8601_3.Data_In <-> KL8601 - 3/Data In
//     PlcTask Inputs/GVL_iXlinker.EtherCAT_Master_BKCUCX.TcTerminals210_EK1100_2.TcTerminals210_2BK1250.A_0039_KL_8610_5_Ch_Adapter_KL8601.KL8601_4.Data_In <-> KL8601 - 4/Data In
//     PlcTask Inputs/GVL_iXlinker.EtherCAT_Master_BKCUCX.TcTerminals210_EK1100_2.TcTerminals210_2BK1250.A_0039_KL_8610_5_Ch_Adapter_KL8601.KL8601_5.Data_In <-> KL8601 - 5/Data In
//     PlcTask Outputs/GVL_iXlinker.EtherCAT_Master_BKCUCX.TcTerminals210_EK1100_2.TcTerminals210_2BK1250.A_0039_KL_8610_5_Ch_Adapter_KL8601.KL8601_1.Ctrl <-> KL8601 - 1/Ctrl
//     PlcTask Outputs/GVL_iXlinker.EtherCAT_Master_BKCUCX.TcTerminals210_EK1100_2.TcTerminals210_2BK1250.A_0039_KL_8610_5_Ch_Adapter_KL8601.KL8601_2.Ctrl <-> KL8601 - 2/Ctrl
//     PlcTask Outputs/GVL_iXlinker.EtherCAT_Master_BKCUCX.TcTerminals210_EK1100_2.TcTerminals210_2BK1250.A_0039_KL_8610_5_Ch_Adapter_KL8601.KL8601_3.Ctrl <-> KL8601 - 3/Ctrl
//     PlcTask Outputs/GVL_iXlinker.EtherCAT_Master_BKCUCX.TcTerminals210_EK1100_2.TcTerminals210_2BK1250.A_0039_KL_8610_5_Ch_Adapter_KL8601.KL8601_4.Ctrl <-> KL8601 - 4/Ctrl
//     PlcTask Outputs/GVL_iXlinker.EtherCAT_Master_BKCUCX.TcTerminals210_EK1100_2.TcTerminals210_2BK1250.A_0039_KL_8610_5_Ch_Adapter_KL8601.KL8601_5.Ctrl <-> KL8601 - 5/Ctrl
//     PlcTask Outputs/GVL_iXlinker.EtherCAT_Master_BKCUCX.TcTerminals210_EK1100_2.TcTerminals210_2BK1250.A_0039_KL_8610_5_Ch_Adapter_KL8601.KL8601_1.Data_Out <-> KL8601 - 1/Data Out
//     PlcTask Outputs/GVL_iXlinker.EtherCAT_Master_BKCUCX.TcTerminals210_EK1100_2.TcTerminals210_2BK1250.A_0039_KL_8610_5_Ch_Adapter_KL8601.KL8601_2.Data_Out <-> KL8601 - 2/Data Out
//     PlcTask Outputs/GVL_iXlinker.EtherCAT_Master_BKCUCX.TcTerminals210_EK1100_2.TcTerminals210_2BK1250.A_0039_KL_8610_5_Ch_Adapter_KL8601.KL8601_3.Data_Out <-> KL8601 - 3/Data Out
//     PlcTask Outputs/GVL_iXlinker.EtherCAT_Master_BKCUCX.TcTerminals210_EK1100_2.TcTerminals210_2BK1250.A_0039_KL_8610_5_Ch_Adapter_KL8601.KL8601_4.Data_Out <-> KL8601 - 4/Data Out
//     PlcTask Outputs/GVL_iXlinker.EtherCAT_Master_BKCUCX.TcTerminals210_EK1100_2.TcTerminals210_2BK1250.A_0039_KL_8610_5_Ch_Adapter_KL8601.KL8601_5.Data_Out <-> KL8601 - 5/Data Out
//   PLC/PLC Instance <-> EtherCAT Master BKCUCX/TcTerminals210_EK1100_2/TcTerminals210_2BK1250/A_0040(KL 8610, 6 Ch. Adapter KL8601)
//     PlcTask Inputs/GVL_iXlinker.EtherCAT_Master_BKCUCX.TcTerminals210_EK1100_2.TcTerminals210_2BK1250.A_0040_KL_8610_6_Ch_Adapter_KL8601.KL8601_1.State <-> KL8601 - 1/State
//     PlcTask Inputs/GVL_iXlinker.EtherCAT_Master_BKCUCX.TcTerminals210_EK1100_2.TcTerminals210_2BK1250.A_0040_KL_8610_6_Ch_Adapter_KL8601.KL8601_2.State <-> KL8601 - 2/State
//     PlcTask Inputs/GVL_iXlinker.EtherCAT_Master_BKCUCX.TcTerminals210_EK1100_2.TcTerminals210_2BK1250.A_0040_KL_8610_6_Ch_Adapter_KL8601.KL8601_3.State <-> KL8601 - 3/State
//     PlcTask Inputs/GVL_iXlinker.EtherCAT_Master_BKCUCX.TcTerminals210_EK1100_2.TcTerminals210_2BK1250.A_0040_KL_8610_6_Ch_Adapter_KL8601.KL8601_4.State <-> KL8601 - 4/State
//     PlcTask Inputs/GVL_iXlinker.EtherCAT_Master_BKCUCX.TcTerminals210_EK1100_2.TcTerminals210_2BK1250.A_0040_KL_8610_6_Ch_Adapter_KL8601.KL8601_5.State <-> KL8601 - 5/State
//     PlcTask Inputs/GVL_iXlinker.EtherCAT_Master_BKCUCX.TcTerminals210_EK1100_2.TcTerminals210_2BK1250.A_0040_KL_8610_6_Ch_Adapter_KL8601.KL8601_6.State <-> KL8601 - 6/State
//     PlcTask Inputs/GVL_iXlinker.EtherCAT_Master_BKCUCX.TcTerminals210_EK1100_2.TcTerminals210_2BK1250.A_0040_KL_8610_6_Ch_Adapter_KL8601.KL8601_1.Data_In <-> KL8601 - 1/Data In
//     PlcTask Inputs/GVL_iXlinker.EtherCAT_Master_BKCUCX.TcTerminals210_EK1100_2.TcTerminals210_2BK1250.A_0040_KL_8610_6_Ch_Adapter_KL8601.KL8601_2.Data_In <-> KL8601 - 2/Data In
//     PlcTask Inputs/GVL_iXlinker.EtherCAT_Master_BKCUCX.TcTerminals210_EK1100_2.TcTerminals210_2BK1250.A_0040_KL_8610_6_Ch_Adapter_KL8601.KL8601_3.Data_In <-> KL8601 - 3/Data In
//     PlcTask Inputs/GVL_iXlinker.EtherCAT_Master_BKCUCX.TcTerminals210_EK1100_2.TcTerminals210_2BK1250.A_0040_KL_8610_6_Ch_Adapter_KL8601.KL8601_4.Data_In <-> KL8601 - 4/Data In
//     PlcTask Inputs/GVL_iXlinker.EtherCAT_Master_BKCUCX.TcTerminals210_EK1100_2.TcTerminals210_2BK1250.A_0040_KL_8610_6_Ch_Adapter_KL8601.KL8601_5.Data_In <-> KL8601 - 5/Data In
//     PlcTask Inputs/GVL_iXlinker.EtherCAT_Master_BKCUCX.TcTerminals210_EK1100_2.TcTerminals210_2BK1250.A_0040_KL_8610_6_Ch_Adapter_KL8601.KL8601_6.Data_In <-> KL8601 - 6/Data In
//     PlcTask Outputs/GVL_iXlinker.EtherCAT_Master_BKCUCX.TcTerminals210_EK1100_2.TcTerminals210_2BK1250.A_0040_KL_8610_6_Ch_Adapter_KL8601.KL8601_1.Ctrl <-> KL8601 - 1/Ctrl
//     PlcTask Outputs/GVL_iXlinker.EtherCAT_Master_BKCUCX.TcTerminals210_EK1100_2.TcTerminals210_2BK1250.A_0040_KL_8610_6_Ch_Adapter_KL8601.KL8601_2.Ctrl <-> KL8601 - 2/Ctrl
//     PlcTask Outputs/GVL_iXlinker.EtherCAT_Master_BKCUCX.TcTerminals210_EK1100_2.TcTerminals210_2BK1250.A_0040_KL_8610_6_Ch_Adapter_KL8601.KL8601_3.Ctrl <-> KL8601 - 3/Ctrl
//     PlcTask Outputs/GVL_iXlinker.EtherCAT_Master_BKCUCX.TcTerminals210_EK1100_2.TcTerminals210_2BK1250.A_0040_KL_8610_6_Ch_Adapter_KL8601.KL8601_4.Ctrl <-> KL8601 - 4/Ctrl
//     PlcTask Outputs/GVL_iXlinker.EtherCAT_Master_BKCUCX.TcTerminals210_EK1100_2.TcTerminals210_2BK1250.A_0040_KL_8610_6_Ch_Adapter_KL8601.KL8601_5.Ctrl <-> KL8601 - 5/Ctrl
//     PlcTask Outputs/GVL_iXlinker.EtherCAT_Master_BKCUCX.TcTerminals210_EK1100_2.TcTerminals210_2BK1250.A_0040_KL_8610_6_Ch_Adapter_KL8601.KL8601_6.Ctrl <-> KL8601 - 6/Ctrl
//     PlcTask Outputs/GVL_iXlinker.EtherCAT_Master_BKCUCX.TcTerminals210_EK1100_2.TcTerminals210_2BK1250.A_0040_KL_8610_6_Ch_Adapter_KL8601.KL8601_1.Data_Out <-> KL8601 - 1/Data Out
//     PlcTask Outputs/GVL_iXlinker.EtherCAT_Master_BKCUCX.TcTerminals210_EK1100_2.TcTerminals210_2BK1250.A_0040_KL_8610_6_Ch_Adapter_KL8601.KL8601_2.Data_Out <-> KL8601 - 2/Data Out
//     PlcTask Outputs/GVL_iXlinker.EtherCAT_Master_BKCUCX.TcTerminals210_EK1100_2.TcTerminals210_2BK1250.A_0040_KL_8610_6_Ch_Adapter_KL8601.KL8601_3.Data_Out <-> KL8601 - 3/Data Out
//     PlcTask Outputs/GVL_iXlinker.EtherCAT_Master_BKCUCX.TcTerminals210_EK1100_2.TcTerminals210_2BK1250.A_0040_KL_8610_6_Ch_Adapter_KL8601.KL8601_4.Data_Out <-> KL8601 - 4/Data Out
//     PlcTask Outputs/GVL_iXlinker.EtherCAT_Master_BKCUCX.TcTerminals210_EK1100_2.TcTerminals210_2BK1250.A_0040_KL_8610_6_Ch_Adapter_KL8601.KL8601_5.Data_Out <-> KL8601 - 5/Data Out
//     PlcTask Outputs/GVL_iXlinker.EtherCAT_Master_BKCUCX.TcTerminals210_EK1100_2.TcTerminals210_2BK1250.A_0040_KL_8610_6_Ch_Adapter_KL8601.KL8601_6.Data_Out <-> KL8601 - 6/Data Out
//   PLC/PLC Instance <-> EtherCAT Master BKCUCX/TcTerminals210_EK1100_2/TcTerminals210_2BK1250/A_0041(KL 8610, 7 Ch. Adapter KL8601)
//     PlcTask Inputs/GVL_iXlinker.EtherCAT_Master_BKCUCX.TcTerminals210_EK1100_2.TcTerminals210_2BK1250.A_0041_KL_8610_7_Ch_Adapter_KL8601.KL8601_1.State <-> KL8601 - 1/State
//     PlcTask Inputs/GVL_iXlinker.EtherCAT_Master_BKCUCX.TcTerminals210_EK1100_2.TcTerminals210_2BK1250.A_0041_KL_8610_7_Ch_Adapter_KL8601.KL8601_2.State <-> KL8601 - 2/State
//     PlcTask Inputs/GVL_iXlinker.EtherCAT_Master_BKCUCX.TcTerminals210_EK1100_2.TcTerminals210_2BK1250.A_0041_KL_8610_7_Ch_Adapter_KL8601.KL8601_3.State <-> KL8601 - 3/State
//     PlcTask Inputs/GVL_iXlinker.EtherCAT_Master_BKCUCX.TcTerminals210_EK1100_2.TcTerminals210_2BK1250.A_0041_KL_8610_7_Ch_Adapter_KL8601.KL8601_4.State <-> KL8601 - 4/State
//     PlcTask Inputs/GVL_iXlinker.EtherCAT_Master_BKCUCX.TcTerminals210_EK1100_2.TcTerminals210_2BK1250.A_0041_KL_8610_7_Ch_Adapter_KL8601.KL8601_5.State <-> KL8601 - 5/State
//     PlcTask Inputs/GVL_iXlinker.EtherCAT_Master_BKCUCX.TcTerminals210_EK1100_2.TcTerminals210_2BK1250.A_0041_KL_8610_7_Ch_Adapter_KL8601.KL8601_6.State <-> KL8601 - 6/State
//     PlcTask Inputs/GVL_iXlinker.EtherCAT_Master_BKCUCX.TcTerminals210_EK1100_2.TcTerminals210_2BK1250.A_0041_KL_8610_7_Ch_Adapter_KL8601.KL8601_7.State <-> KL8601 - 7/State
//     PlcTask Inputs/GVL_iXlinker.EtherCAT_Master_BKCUCX.TcTerminals210_EK1100_2.TcTerminals210_2BK1250.A_0041_KL_8610_7_Ch_Adapter_KL8601.KL8601_1.Data_In <-> KL8601 - 1/Data In
//     PlcTask Inputs/GVL_iXlinker.EtherCAT_Master_BKCUCX.TcTerminals210_EK1100_2.TcTerminals210_2BK1250.A_0041_KL_8610_7_Ch_Adapter_KL8601.KL8601_2.Data_In <-> KL8601 - 2/Data In
//     PlcTask Inputs/GVL_iXlinker.EtherCAT_Master_BKCUCX.TcTerminals210_EK1100_2.TcTerminals210_2BK1250.A_0041_KL_8610_7_Ch_Adapter_KL8601.KL8601_3.Data_In <-> KL8601 - 3/Data In
//     PlcTask Inputs/GVL_iXlinker.EtherCAT_Master_BKCUCX.TcTerminals210_EK1100_2.TcTerminals210_2BK1250.A_0041_KL_8610_7_Ch_Adapter_KL8601.KL8601_4.Data_In <-> KL8601 - 4/Data In
//     PlcTask Inputs/GVL_iXlinker.EtherCAT_Master_BKCUCX.TcTerminals210_EK1100_2.TcTerminals210_2BK1250.A_0041_KL_8610_7_Ch_Adapter_KL8601.KL8601_5.Data_In <-> KL8601 - 5/Data In
//     PlcTask Inputs/GVL_iXlinker.EtherCAT_Master_BKCUCX.TcTerminals210_EK1100_2.TcTerminals210_2BK1250.A_0041_KL_8610_7_Ch_Adapter_KL8601.KL8601_6.Data_In <-> KL8601 - 6/Data In
//     PlcTask Inputs/GVL_iXlinker.EtherCAT_Master_BKCUCX.TcTerminals210_EK1100_2.TcTerminals210_2BK1250.A_0041_KL_8610_7_Ch_Adapter_KL8601.KL8601_7.Data_In <-> KL8601 - 7/Data In
//     PlcTask Outputs/GVL_iXlinker.EtherCAT_Master_BKCUCX.TcTerminals210_EK1100_2.TcTerminals210_2BK1250.A_0041_KL_8610_7_Ch_Adapter_KL8601.KL8601_1.Ctrl <-> KL8601 - 1/Ctrl
//     PlcTask Outputs/GVL_iXlinker.EtherCAT_Master_BKCUCX.TcTerminals210_EK1100_2.TcTerminals210_2BK1250.A_0041_KL_8610_7_Ch_Adapter_KL8601.KL8601_2.Ctrl <-> KL8601 - 2/Ctrl
//     PlcTask Outputs/GVL_iXlinker.EtherCAT_Master_BKCUCX.TcTerminals210_EK1100_2.TcTerminals210_2BK1250.A_0041_KL_8610_7_Ch_Adapter_KL8601.KL8601_3.Ctrl <-> KL8601 - 3/Ctrl
//     PlcTask Outputs/GVL_iXlinker.EtherCAT_Master_BKCUCX.TcTerminals210_EK1100_2.TcTerminals210_2BK1250.A_0041_KL_8610_7_Ch_Adapter_KL8601.KL8601_4.Ctrl <-> KL8601 - 4/Ctrl
//     PlcTask Outputs/GVL_iXlinker.EtherCAT_Master_BKCUCX.TcTerminals210_EK1100_2.TcTerminals210_2BK1250.A_0041_KL_8610_7_Ch_Adapter_KL8601.KL8601_5.Ctrl <-> KL8601 - 5/Ctrl
//     PlcTask Outputs/GVL_iXlinker.EtherCAT_Master_BKCUCX.TcTerminals210_EK1100_2.TcTerminals210_2BK1250.A_0041_KL_8610_7_Ch_Adapter_KL8601.KL8601_6.Ctrl <-> KL8601 - 6/Ctrl
//     PlcTask Outputs/GVL_iXlinker.EtherCAT_Master_BKCUCX.TcTerminals210_EK1100_2.TcTerminals210_2BK1250.A_0041_KL_8610_7_Ch_Adapter_KL8601.KL8601_7.Ctrl <-> KL8601 - 7/Ctrl
//     PlcTask Outputs/GVL_iXlinker.EtherCAT_Master_BKCUCX.TcTerminals210_EK1100_2.TcTerminals210_2BK1250.A_0041_KL_8610_7_Ch_Adapter_KL8601.KL8601_1.Data_Out <-> KL8601 - 1/Data Out
//     PlcTask Outputs/GVL_iXlinker.EtherCAT_Master_BKCUCX.TcTerminals210_EK1100_2.TcTerminals210_2BK1250.A_0041_KL_8610_7_Ch_Adapter_KL8601.KL8601_2.Data_Out <-> KL8601 - 2/Data Out
//     PlcTask Outputs/GVL_iXlinker.EtherCAT_Master_BKCUCX.TcTerminals210_EK1100_2.TcTerminals210_2BK1250.A_0041_KL_8610_7_Ch_Adapter_KL8601.KL8601_3.Data_Out <-> KL8601 - 3/Data Out
//     PlcTask Outputs/GVL_iXlinker.EtherCAT_Master_BKCUCX.TcTerminals210_EK1100_2.TcTerminals210_2BK1250.A_0041_KL_8610_7_Ch_Adapter_KL8601.KL8601_4.Data_Out <-> KL8601 - 4/Data Out
//     PlcTask Outputs/GVL_iXlinker.EtherCAT_Master_BKCUCX.TcTerminals210_EK1100_2.TcTerminals210_2BK1250.A_0041_KL_8610_7_Ch_Adapter_KL8601.KL8601_5.Data_Out <-> KL8601 - 5/Data Out
//     PlcTask Outputs/GVL_iXlinker.EtherCAT_Master_BKCUCX.TcTerminals210_EK1100_2.TcTerminals210_2BK1250.A_0041_KL_8610_7_Ch_Adapter_KL8601.KL8601_6.Data_Out <-> KL8601 - 6/Data Out
//     PlcTask Outputs/GVL_iXlinker.EtherCAT_Master_BKCUCX.TcTerminals210_EK1100_2.TcTerminals210_2BK1250.A_0041_KL_8610_7_Ch_Adapter_KL8601.KL8601_7.Data_Out <-> KL8601 - 7/Data Out
//   PLC/PLC Instance <-> EtherCAT Master BKCUCX/TcTerminals210_EK1100_2/TcTerminals210_2BK1250/A_0042(KL 8610, 8 Ch. Adapter KL8601)
//     PlcTask Inputs/GVL_iXlinker.EtherCAT_Master_BKCUCX.TcTerminals210_EK1100_2.TcTerminals210_2BK1250.A_0042_KL_8610_8_Ch_Adapter_KL8601.KL8601_1.State <-> KL8601 - 1/State
//     PlcTask Inputs/GVL_iXlinker.EtherCAT_Master_BKCUCX.TcTerminals210_EK1100_2.TcTerminals210_2BK1250.A_0042_KL_8610_8_Ch_Adapter_KL8601.KL8601_2.State <-> KL8601 - 2/State
//     PlcTask Inputs/GVL_iXlinker.EtherCAT_Master_BKCUCX.TcTerminals210_EK1100_2.TcTerminals210_2BK1250.A_0042_KL_8610_8_Ch_Adapter_KL8601.KL8601_3.State <-> KL8601 - 3/State
//     PlcTask Inputs/GVL_iXlinker.EtherCAT_Master_BKCUCX.TcTerminals210_EK1100_2.TcTerminals210_2BK1250.A_0042_KL_8610_8_Ch_Adapter_KL8601.KL8601_4.State <-> KL8601 - 4/State
//     PlcTask Inputs/GVL_iXlinker.EtherCAT_Master_BKCUCX.TcTerminals210_EK1100_2.TcTerminals210_2BK1250.A_0042_KL_8610_8_Ch_Adapter_KL8601.KL8601_5.State <-> KL8601 - 5/State
//     PlcTask Inputs/GVL_iXlinker.EtherCAT_Master_BKCUCX.TcTerminals210_EK1100_2.TcTerminals210_2BK1250.A_0042_KL_8610_8_Ch_Adapter_KL8601.KL8601_6.State <-> KL8601 - 6/State
//     PlcTask Inputs/GVL_iXlinker.EtherCAT_Master_BKCUCX.TcTerminals210_EK1100_2.TcTerminals210_2BK1250.A_0042_KL_8610_8_Ch_Adapter_KL8601.KL8601_7.State <-> KL8601 - 7/State
//     PlcTask Inputs/GVL_iXlinker.EtherCAT_Master_BKCUCX.TcTerminals210_EK1100_2.TcTerminals210_2BK1250.A_0042_KL_8610_8_Ch_Adapter_KL8601.KL8601_8.State <-> KL8601 - 8/State
//     PlcTask Inputs/GVL_iXlinker.EtherCAT_Master_BKCUCX.TcTerminals210_EK1100_2.TcTerminals210_2BK1250.A_0042_KL_8610_8_Ch_Adapter_KL8601.KL8601_1.Data_In <-> KL8601 - 1/Data In
//     PlcTask Inputs/GVL_iXlinker.EtherCAT_Master_BKCUCX.TcTerminals210_EK1100_2.TcTerminals210_2BK1250.A_0042_KL_8610_8_Ch_Adapter_KL8601.KL8601_2.Data_In <-> KL8601 - 2/Data In
//     PlcTask Inputs/GVL_iXlinker.EtherCAT_Master_BKCUCX.TcTerminals210_EK1100_2.TcTerminals210_2BK1250.A_0042_KL_8610_8_Ch_Adapter_KL8601.KL8601_3.Data_In <-> KL8601 - 3/Data In
//     PlcTask Inputs/GVL_iXlinker.EtherCAT_Master_BKCUCX.TcTerminals210_EK1100_2.TcTerminals210_2BK1250.A_0042_KL_8610_8_Ch_Adapter_KL8601.KL8601_4.Data_In <-> KL8601 - 4/Data In
//     PlcTask Inputs/GVL_iXlinker.EtherCAT_Master_BKCUCX.TcTerminals210_EK1100_2.TcTerminals210_2BK1250.A_0042_KL_8610_8_Ch_Adapter_KL8601.KL8601_5.Data_In <-> KL8601 - 5/Data In
//     PlcTask Inputs/GVL_iXlinker.EtherCAT_Master_BKCUCX.TcTerminals210_EK1100_2.TcTerminals210_2BK1250.A_0042_KL_8610_8_Ch_Adapter_KL8601.KL8601_6.Data_In <-> KL8601 - 6/Data In
//     PlcTask Inputs/GVL_iXlinker.EtherCAT_Master_BKCUCX.TcTerminals210_EK1100_2.TcTerminals210_2BK1250.A_0042_KL_8610_8_Ch_Adapter_KL8601.KL8601_7.Data_In <-> KL8601 - 7/Data In
//     PlcTask Inputs/GVL_iXlinker.EtherCAT_Master_BKCUCX.TcTerminals210_EK1100_2.TcTerminals210_2BK1250.A_0042_KL_8610_8_Ch_Adapter_KL8601.KL8601_8.Data_In <-> KL8601 - 8/Data In
//     PlcTask Outputs/GVL_iXlinker.EtherCAT_Master_BKCUCX.TcTerminals210_EK1100_2.TcTerminals210_2BK1250.A_0042_KL_8610_8_Ch_Adapter_KL8601.KL8601_1.Ctrl <-> KL8601 - 1/Ctrl
//     PlcTask Outputs/GVL_iXlinker.EtherCAT_Master_BKCUCX.TcTerminals210_EK1100_2.TcTerminals210_2BK1250.A_0042_KL_8610_8_Ch_Adapter_KL8601.KL8601_2.Ctrl <-> KL8601 - 2/Ctrl
//     PlcTask Outputs/GVL_iXlinker.EtherCAT_Master_BKCUCX.TcTerminals210_EK1100_2.TcTerminals210_2BK1250.A_0042_KL_8610_8_Ch_Adapter_KL8601.KL8601_3.Ctrl <-> KL8601 - 3/Ctrl
//     PlcTask Outputs/GVL_iXlinker.EtherCAT_Master_BKCUCX.TcTerminals210_EK1100_2.TcTerminals210_2BK1250.A_0042_KL_8610_8_Ch_Adapter_KL8601.KL8601_4.Ctrl <-> KL8601 - 4/Ctrl
//     PlcTask Outputs/GVL_iXlinker.EtherCAT_Master_BKCUCX.TcTerminals210_EK1100_2.TcTerminals210_2BK1250.A_0042_KL_8610_8_Ch_Adapter_KL8601.KL8601_5.Ctrl <-> KL8601 - 5/Ctrl
//     PlcTask Outputs/GVL_iXlinker.EtherCAT_Master_BKCUCX.TcTerminals210_EK1100_2.TcTerminals210_2BK1250.A_0042_KL_8610_8_Ch_Adapter_KL8601.KL8601_6.Ctrl <-> KL8601 - 6/Ctrl
//     PlcTask Outputs/GVL_iXlinker.EtherCAT_Master_BKCUCX.TcTerminals210_EK1100_2.TcTerminals210_2BK1250.A_0042_KL_8610_8_Ch_Adapter_KL8601.KL8601_7.Ctrl <-> KL8601 - 7/Ctrl
//     PlcTask Outputs/GVL_iXlinker.EtherCAT_Master_BKCUCX.TcTerminals210_EK1100_2.TcTerminals210_2BK1250.A_0042_KL_8610_8_Ch_Adapter_KL8601.KL8601_8.Ctrl <-> KL8601 - 8/Ctrl
//     PlcTask Outputs/GVL_iXlinker.EtherCAT_Master_BKCUCX.TcTerminals210_EK1100_2.TcTerminals210_2BK1250.A_0042_KL_8610_8_Ch_Adapter_KL8601.KL8601_1.Data_Out <-> KL8601 - 1/Data Out
//     PlcTask Outputs/GVL_iXlinker.EtherCAT_Master_BKCUCX.TcTerminals210_EK1100_2.TcTerminals210_2BK1250.A_0042_KL_8610_8_Ch_Adapter_KL8601.KL8601_2.Data_Out <-> KL8601 - 2/Data Out
//     PlcTask Outputs/GVL_iXlinker.EtherCAT_Master_BKCUCX.TcTerminals210_EK1100_2.TcTerminals210_2BK1250.A_0042_KL_8610_8_Ch_Adapter_KL8601.KL8601_3.Data_Out <-> KL8601 - 3/Data Out
//     PlcTask Outputs/GVL_iXlinker.EtherCAT_Master_BKCUCX.TcTerminals210_EK1100_2.TcTerminals210_2BK1250.A_0042_KL_8610_8_Ch_Adapter_KL8601.KL8601_4.Data_Out <-> KL8601 - 4/Data Out
//     PlcTask Outputs/GVL_iXlinker.EtherCAT_Master_BKCUCX.TcTerminals210_EK1100_2.TcTerminals210_2BK1250.A_0042_KL_8610_8_Ch_Adapter_KL8601.KL8601_5.Data_Out <-> KL8601 - 5/Data Out
//     PlcTask Outputs/GVL_iXlinker.EtherCAT_Master_BKCUCX.TcTerminals210_EK1100_2.TcTerminals210_2BK1250.A_0042_KL_8610_8_Ch_Adapter_KL8601.KL8601_6.Data_Out <-> KL8601 - 6/Data Out
//     PlcTask Outputs/GVL_iXlinker.EtherCAT_Master_BKCUCX.TcTerminals210_EK1100_2.TcTerminals210_2BK1250.A_0042_KL_8610_8_Ch_Adapter_KL8601.KL8601_7.Data_Out <-> KL8601 - 7/Data Out
//     PlcTask Outputs/GVL_iXlinker.EtherCAT_Master_BKCUCX.TcTerminals210_EK1100_2.TcTerminals210_2BK1250.A_0042_KL_8610_8_Ch_Adapter_KL8601.KL8601_8.Data_Out <-> KL8601 - 8/Data Out
//   PLC/PLC Instance <-> EtherCAT Master BKCUCX/TcTerminals210_EK1100_2/TcTerminals210_2BK1250/A_0050(KL 9110, Power Supplier with LED and Diag. (24V))
//     PlcTask Inputs/GVL_iXlinker.EtherCAT_Master_BKCUCX.TcTerminals210_EK1100_2.TcTerminals210_2BK1250.A_0050_KL_9110_Power_Supplier_with_LED_and_Diag_24V.Channel_1.Power <-> Channel 1/Power
//     PlcTask Inputs/GVL_iXlinker.EtherCAT_Master_BKCUCX.TcTerminals210_EK1100_2.TcTerminals210_2BK1250.A_0050_KL_9110_Power_Supplier_with_LED_and_Diag_24V.Channel_1.ShortCircuit <-> Channel 1/ShortCircuit
//   PLC/PLC Instance <-> EtherCAT Master BKCUCX/TcTerminals210_EK1100_2/TcTerminals210_2BK1250/A_0052(KL 9160, Power Supplier with LED and Diag. (230V))
//     PlcTask Inputs/GVL_iXlinker.EtherCAT_Master_BKCUCX.TcTerminals210_EK1100_2.TcTerminals210_2BK1250.A_0052_KL_9160_Power_Supplier_with_LED_and_Diag_230V.Channel_1.Power <-> Channel 1/Power
//     PlcTask Inputs/GVL_iXlinker.EtherCAT_Master_BKCUCX.TcTerminals210_EK1100_2.TcTerminals210_2BK1250.A_0052_KL_9160_Power_Supplier_with_LED_and_Diag_230V.Channel_1.ShortCircuit <-> Channel 1/ShortCircuit
//   PLC/PLC Instance <-> EtherCAT Master BKCUCX/TcTerminals210_EK1100_2/TcTerminals210_2BK1250/A_0064(KL 9191 Dig I/O)
//     PlcTask Inputs/GVL_iXlinker.EtherCAT_Master_BKCUCX.TcTerminals210_EK1100_2.TcTerminals210_2BK1250.A_0064_KL_9191_Dig_I_O.Channel_1.Contact_DI1 <-> Channel 1/Contact DI1
//     PlcTask Inputs/GVL_iXlinker.EtherCAT_Master_BKCUCX.TcTerminals210_EK1100_2.TcTerminals210_2BK1250.A_0064_KL_9191_Dig_I_O.Channel_1.Contact_DI2 <-> Channel 1/Contact DI2
//     PlcTask Inputs/GVL_iXlinker.EtherCAT_Master_BKCUCX.TcTerminals210_EK1100_2.TcTerminals210_2BK1250.A_0064_KL_9191_Dig_I_O.Channel_1.Contact_DI3 <-> Channel 1/Contact DI3
//     PlcTask Outputs/GVL_iXlinker.EtherCAT_Master_BKCUCX.TcTerminals210_EK1100_2.TcTerminals210_2BK1250.A_0064_KL_9191_Dig_I_O.Channel_1.LED_DO1 <-> Channel 1/LED DO1
//     PlcTask Outputs/GVL_iXlinker.EtherCAT_Master_BKCUCX.TcTerminals210_EK1100_2.TcTerminals210_2BK1250.A_0064_KL_9191_Dig_I_O.Channel_1.Relay_2kW <-> Channel 1/Relay 2kW
//     PlcTask Outputs/GVL_iXlinker.EtherCAT_Master_BKCUCX.TcTerminals210_EK1100_2.TcTerminals210_2BK1250.A_0064_KL_9191_Dig_I_O.Channel_1.Relay_FAN1 <-> Channel 1/Relay FAN1
//     PlcTask Outputs/GVL_iXlinker.EtherCAT_Master_BKCUCX.TcTerminals210_EK1100_2.TcTerminals210_2BK1250.A_0064_KL_9191_Dig_I_O.Channel_1.Relay_FAN2 <-> Channel 1/Relay FAN2
//     PlcTask Outputs/GVL_iXlinker.EtherCAT_Master_BKCUCX.TcTerminals210_EK1100_2.TcTerminals210_2BK1250.A_0064_KL_9191_Dig_I_O.Channel_1.Relay_FAN3 <-> Channel 1/Relay FAN3
//     PlcTask Outputs/GVL_iXlinker.EtherCAT_Master_BKCUCX.TcTerminals210_EK1100_2.TcTerminals210_2BK1250.A_0064_KL_9191_Dig_I_O.Channel_1.TRIAC_Y1 <-> Channel 1/TRIAC Y1
//     PlcTask Outputs/GVL_iXlinker.EtherCAT_Master_BKCUCX.TcTerminals210_EK1100_2.TcTerminals210_2BK1250.A_0064_KL_9191_Dig_I_O.Channel_1.TRIAC_Y2 <-> Channel 1/TRIAC Y2
//   PLC/PLC Instance <-> EtherCAT Master BKCUCX/TcTerminals210_EK1100_2/TcTerminals210_2BK1250/A_0067(KL 9210, Power Supplier with Fuse, LED and Diag. (24V))
//     PlcTask Inputs/GVL_iXlinker.EtherCAT_Master_BKCUCX.TcTerminals210_EK1100_2.TcTerminals210_2BK1250.A_0067_KL_9210_Power_Supplier_with_Fuse_LED_and_Diag_24V.Channel_1.Power <-> Channel 1/Power
//     PlcTask Inputs/GVL_iXlinker.EtherCAT_Master_BKCUCX.TcTerminals210_EK1100_2.TcTerminals210_2BK1250.A_0067_KL_9210_Power_Supplier_with_Fuse_LED_and_Diag_24V.Channel_1.ShortCircuit <-> Channel 1/ShortCircuit
//   PLC/PLC Instance <-> EtherCAT Master BKCUCX/TcTerminals210_EK1100_2/TcTerminals210_2BK1250/A_0069(KL 9260, Power Supplier with Fuse, LED and Diag. (230V))
//     PlcTask Inputs/GVL_iXlinker.EtherCAT_Master_BKCUCX.TcTerminals210_EK1100_2.TcTerminals210_2BK1250.A_0069_KL_9260_Power_Supplier_with_Fuse_LED_and_Diag_230V.Channel_1.Power <-> Channel 1/Power
//     PlcTask Inputs/GVL_iXlinker.EtherCAT_Master_BKCUCX.TcTerminals210_EK1100_2.TcTerminals210_2BK1250.A_0069_KL_9260_Power_Supplier_with_Fuse_LED_and_Diag_230V.Channel_1.ShortCircuit <-> Channel 1/ShortCircuit
//   PLC/PLC Instance <-> EtherCAT Master BKCUCX/TcTerminals210_EK1100_2/TcTerminals210_2BK1250/A_0078(KL 9505-0010, Power Supplier 5V, 0.5A, Diag)
//     PlcTask Inputs/GVL_iXlinker.EtherCAT_Master_BKCUCX.TcTerminals210_EK1100_2.TcTerminals210_2BK1250.A_0078_KL_9505_0010_Power_Supplier_5V_0_5A_Diag.Diag_1.Supply_Voltage_OK <-> Diag 1/Supply Voltage OK
//     PlcTask Inputs/GVL_iXlinker.EtherCAT_Master_BKCUCX.TcTerminals210_EK1100_2.TcTerminals210_2BK1250.A_0078_KL_9505_0010_Power_Supplier_5V_0_5A_Diag.Diag_1.Over_current <-> Diag 1/Over current
//   PLC/PLC Instance <-> EtherCAT Master BKCUCX/TcTerminals210_EK1100_2/TcTerminals210_2BK1250/A_0080(KL 9508-0010, Power Supplier 8V, 0.5A, Diag)
//     PlcTask Inputs/GVL_iXlinker.EtherCAT_Master_BKCUCX.TcTerminals210_EK1100_2.TcTerminals210_2BK1250.A_0080_KL_9508_0010_Power_Supplier_8V_0_5A_Diag.Diag_1.Supply_Voltage_OK <-> Diag 1/Supply Voltage OK
//     PlcTask Inputs/GVL_iXlinker.EtherCAT_Master_BKCUCX.TcTerminals210_EK1100_2.TcTerminals210_2BK1250.A_0080_KL_9508_0010_Power_Supplier_8V_0_5A_Diag.Diag_1.Over_current <-> Diag 1/Over current
//   PLC/PLC Instance <-> EtherCAT Master BKCUCX/TcTerminals210_EK1100_2/TcTerminals210_2BK1250/A_0082(KL 9510-0010, Power Supplier 10V, 0.5A, Diag)
//     PlcTask Inputs/GVL_iXlinker.EtherCAT_Master_BKCUCX.TcTerminals210_EK1100_2.TcTerminals210_2BK1250.A_0082_KL_9510_0010_Power_Supplier_10V_0_5A_Diag.Diag_1.Supply_Voltage_OK <-> Diag 1/Supply Voltage OK
//     PlcTask Inputs/GVL_iXlinker.EtherCAT_Master_BKCUCX.TcTerminals210_EK1100_2.TcTerminals210_2BK1250.A_0082_KL_9510_0010_Power_Supplier_10V_0_5A_Diag.Diag_1.Over_current <-> Diag 1/Over current
//   PLC/PLC Instance <-> EtherCAT Master BKCUCX/TcTerminals210_EK1100_2/TcTerminals210_2BK1250/A_0084(KL 9512-0010, Power Supplier 12V, 0.5A, Diag)
//     PlcTask Inputs/GVL_iXlinker.EtherCAT_Master_BKCUCX.TcTerminals210_EK1100_2.TcTerminals210_2BK1250.A_0084_KL_9512_0010_Power_Supplier_12V_0_5A_Diag.Diag_1.Supply_Voltage_OK <-> Diag 1/Supply Voltage OK
//     PlcTask Inputs/GVL_iXlinker.EtherCAT_Master_BKCUCX.TcTerminals210_EK1100_2.TcTerminals210_2BK1250.A_0084_KL_9512_0010_Power_Supplier_12V_0_5A_Diag.Diag_1.Over_current <-> Diag 1/Over current
//   PLC/PLC Instance <-> EtherCAT Master BKCUCX/TcTerminals210_EK1100_2/TcTerminals210_2BK1250/A_0086(KL 9515-0010, Power Supplier 15V, 0.5A, Diag)
//     PlcTask Inputs/GVL_iXlinker.EtherCAT_Master_BKCUCX.TcTerminals210_EK1100_2.TcTerminals210_2BK1250.A_0086_KL_9515_0010_Power_Supplier_15V_0_5A_Diag.Diag_1.Supply_Voltage_OK <-> Diag 1/Supply Voltage OK
//     PlcTask Inputs/GVL_iXlinker.EtherCAT_Master_BKCUCX.TcTerminals210_EK1100_2.TcTerminals210_2BK1250.A_0086_KL_9515_0010_Power_Supplier_15V_0_5A_Diag.Diag_1.Over_current <-> Diag 1/Over current
//   PLC/PLC Instance <-> EtherCAT Master BKCUCX/TcTerminals210_EK1100_2/TcTerminals210_2BK1250/A_0087(KL 9528, Power Supplier AS-i, 2A)
//     PlcTask Inputs/GVL_iXlinker.EtherCAT_Master_BKCUCX.TcTerminals210_EK1100_2.TcTerminals210_2BK1250.A_0087_KL_9528_Power_Supplier_AS_i_2A.Channel_1.Overload <-> Channel 1/Overload
//     PlcTask Inputs/GVL_iXlinker.EtherCAT_Master_BKCUCX.TcTerminals210_EK1100_2.TcTerminals210_2BK1250.A_0087_KL_9528_Power_Supplier_AS_i_2A.Channel_1.Undervoltage <-> Channel 1/Undervoltage
//     PlcTask Outputs/GVL_iXlinker.EtherCAT_Master_BKCUCX.TcTerminals210_EK1100_2.TcTerminals210_2BK1250.A_0087_KL_9528_Power_Supplier_AS_i_2A.Channel_1.Reset <-> Channel 1/Reset
//   PLC/PLC Instance <-> EtherCAT Master BKCUCX/TcTerminals210_EK1100_2/TcTerminals210_2BK1250/A_0092(KLWORD (1 In- and 1 Output Word))
//     PlcTask Inputs/GVL_iXlinker.EtherCAT_Master_BKCUCX.TcTerminals210_EK1100_2.TcTerminals210_2BK1250.A_0092_KLWORD_1_In_and_1_Output_Word.Channel_1.VarIn <-> Channel 1/VarIn
//     PlcTask Outputs/GVL_iXlinker.EtherCAT_Master_BKCUCX.TcTerminals210_EK1100_2.TcTerminals210_2BK1250.A_0092_KLWORD_1_In_and_1_Output_Word.Channel_1.VarOut <-> Channel 1/VarOut
//   PLC/PLC Instance <-> EtherCAT_Master_BKCUCX
//     PlcTask Inputs/GVL_iXlinker.EtherCAT_Master_BKCUCX.SyncUnits._default._unreferenced.WcState.WcState <-> SyncUnits/<default>/<unreferenced>/WcState/WcState
//     PlcTask Inputs/GVL_iXlinker.EtherCAT_Master_BKCUCX.SyncUnits._default._unreferenced.InfoData.ObjectId <-> SyncUnits/<default>/<unreferenced>/InfoData/ObjectId
//     PlcTask Inputs/GVL_iXlinker.EtherCAT_Master_BKCUCX.SyncUnits._default._unreferenced.InfoData.State <-> SyncUnits/<default>/<unreferenced>/InfoData/State
//     PlcTask Inputs/GVL_iXlinker.EtherCAT_Master_BKCUCX.SyncUnits._default._unreferenced.InfoData.SlaveCount <-> SyncUnits/<default>/<unreferenced>/InfoData/SlaveCount
//     PlcTask Inputs/GVL_iXlinker.EtherCAT_Master_BKCUCX.SyncUnits._default.PlcTask.WcState.WcState <-> SyncUnits/<default>/PlcTask/WcState/WcState
//     PlcTask Inputs/GVL_iXlinker.EtherCAT_Master_BKCUCX.SyncUnits._default.PlcTask.InfoData.ObjectId <-> SyncUnits/<default>/PlcTask/InfoData/ObjectId
//     PlcTask Inputs/GVL_iXlinker.EtherCAT_Master_BKCUCX.SyncUnits._default.PlcTask.InfoData.State <-> SyncUnits/<default>/PlcTask/InfoData/State
//     PlcTask Inputs/GVL_iXlinker.EtherCAT_Master_BKCUCX.SyncUnits._default.PlcTask.InfoData.SlaveCount <-> SyncUnits/<default>/PlcTask/InfoData/SlaveCount
//     PlcTask Inputs/GVL_iXlinker.EtherCAT_Master_BKCUCX.Inputs.SlaveCount <-> Inputs/SlaveCount
//     PlcTask Inputs/GVL_iXlinker.EtherCAT_Master_BKCUCX.Inputs.DevState <-> Inputs/DevState
//     PlcTask Inputs/GVL_iXlinker.EtherCAT_Master_BKCUCX.Inputs.Frm{0..25}State <-> Inputs/Frm{0..25}State  (26 links)
//     PlcTask Inputs/GVL_iXlinker.EtherCAT_Master_BKCUCX.Inputs.Frm{0..25}WcState <-> Inputs/Frm{0..25}WcState  (26 links)
//     PlcTask Inputs/GVL_iXlinker.EtherCAT_Master_BKCUCX.Inputs.Frm{0..25}InputToggle <-> Inputs/Frm{0..25}InputToggle  (26 links)
//     PlcTask Outputs/GVL_iXlinker.EtherCAT_Master_BKCUCX.Outputs.DevCtrl <-> Outputs/DevCtrl
//     PlcTask Outputs/GVL_iXlinker.EtherCAT_Master_BKCUCX.Outputs.Frm{0..25}Ctrl <-> Outputs/Frm{0..25}Ctrl  (26 links)
//     PlcTask Outputs/GVL_iXlinker.EtherCAT_Master_BKCUCX.Outputs.Frm{0..25}WcCtrl <-> Outputs/Frm{0..25}WcCtrl  (26 links)
//     PlcTask Inputs/GVL_iXlinker.EtherCAT_Master_BKCUCX.InfoData.ChangeCount <-> InfoData/ChangeCount
//     PlcTask Inputs/GVL_iXlinker.EtherCAT_Master_BKCUCX.InfoData.DevId <-> InfoData/DevId
//     PlcTask Inputs/GVL_iXlinker.EtherCAT_Master_BKCUCX.InfoData.AmsNetId <-> InfoData/AmsNetId
//     PlcTask Inputs/GVL_iXlinker.EtherCAT_Master_BKCUCX.InfoData.CfgSlaveCount <-> InfoData/CfgSlaveCount
//     PlcTask Inputs/GVL_iXlinker.EtherCAT_Master_BKCUCX.InfoData.DcToTcTimeOffset <-> InfoData/DcToTcTimeOffset
//     PlcTask Inputs/GVL_iXlinker.EtherCAT_Master_BKCUCX.InfoData.DcToExtTimeOffset <-> InfoData/DcToExtTimeOffset

CONFIGURATION PLC
    RESOURCE PLC ON TwinCAT3
        TASK PlcTask(INTERVAL := T#10ms, PRIORITY := 20);
        PROGRAM MAIN WITH PlcTask : MAIN;
    END_RESOURCE
END_CONFIGURATION

// ---- DUTs/IO/PDOs/InfoData_6F19DB2B.TcDUT
{attribute 'GeneratedUsingTerminal: EK1100-0000-0018'}
{attribute addProperty BoxType "EK1100-0000-0018"}
{attribute addProperty Id "StateAT %I*UINT2"}
{attribute addProperty CRC "1863965483"}
{attribute addProperty Size "2"}
TYPE InfoData_6F19DB2B :
STRUCT
	{attribute addProperty Name "State"}
	State AT %I* : UINT;
END_STRUCT
END_TYPE

// ---- DUTs/IO/PDOs/Inputs_CC16D1F4.TcDUT
{attribute 'GeneratedUsingTerminal: BK1250-0000-0000'}
{attribute addProperty BoxType "BK1250-0000-0000"}
{attribute addProperty Id "CouplerStateAT %I*UINT0"}
{attribute addProperty CRC "3424047604"}
{attribute addProperty Size "0"}
TYPE Inputs_CC16D1F4 EXTENDS InputBase_8311D824 :
STRUCT
	{attribute addProperty Name "CouplerState"}
	CouplerState AT %I* : UINT;
END_STRUCT
END_TYPE

// ---- DUTs/IO/PDOs/Outputs_D8BAB3B3.TcDUT
{attribute 'GeneratedUsingTerminal: BK1250-0000-0000'}
{attribute addProperty BoxType "BK1250-0000-0000"}
{attribute addProperty Id "CouplerCtrlAT %I*UINT0"}
{attribute addProperty CRC "3636114355"}
{attribute addProperty Size "0"}
TYPE Outputs_D8BAB3B3 EXTENDS InputBase_8311D824 :
STRUCT
	{attribute addProperty Name "CouplerCtrl"}
	CouplerCtrl AT %I* : UINT;
END_STRUCT
END_TYPE

// ---- DUTs/IO/PDOs/WcState_9091E0EB.TcDUT
{attribute 'GeneratedUsingTerminal: BK1250-0000-0000'}
{attribute addProperty BoxType "BK1250-0000-0000"}
{attribute addProperty Id "WcStateAT %I*BOOL1InputToggleAT %I*BOOL1"}
{attribute addProperty CRC "2425479403"}
{attribute addProperty Size "2"}
TYPE WcState_9091E0EB :
STRUCT
	{attribute addProperty Name "WcState"}
	WcState AT %I* : BOOL;
	{attribute addProperty Name "InputToggle"}
	InputToggle AT %I* : BOOL;
END_STRUCT
END_TYPE

// ---- DUTs/IO/PDOs/InfoData_90184F0C.TcDUT
{attribute 'GeneratedUsingTerminal: BK1250-0000-0000'}
{attribute addProperty BoxType "BK1250-0000-0000"}
{attribute addProperty Id "AdsAddrAT %I*AMSADDR8AoeNetIdAT %I*AMSNETID6StateAT %I*UINT2"}
{attribute addProperty CRC "2417512204"}
{attribute addProperty Size "16"}
TYPE InfoData_90184F0C EXTENDS InputBase_8311D824 :
STRUCT
	{attribute addProperty Name "AdsAddr"}
	AdsAddr AT %I* : AMSADDR;
	{attribute addProperty Name "AoeNetId"}
	AoeNetId AT %I* : AMSNETID;
	{attribute addProperty Name "State"}
	State AT %I* : UINT;
END_STRUCT
END_TYPE

// ---- DUTs/IO/PDOs/Channel_87C95E76.TcDUT
{attribute 'GeneratedUsingTerminal: KL1002'}
{attribute addProperty BoxType "KL1002"}
{attribute addProperty Id "InputAT %I*BOOL0"}
{attribute addProperty CRC "2278121078"}
{attribute addProperty Size "0"}
TYPE Channel_87C95E76 EXTENDS InputBase_8311D824 :
STRUCT
	{attribute addProperty Name "Input"}
	Input AT %I* : BOOL;
END_STRUCT
END_TYPE

// ---- DUTs/IO/PDOs/InfoData_32EB74EA.TcDUT
{attribute 'GeneratedUsingTerminal: BK1120-0000-0000'}
{attribute addProperty BoxType "BK1120-0000-0000"}
{attribute addProperty Id "AdsAddrAT %I*AMSADDR8StateAT %I*UINT2"}
{attribute addProperty CRC "854291690"}
{attribute addProperty Size "10"}
TYPE InfoData_32EB74EA EXTENDS InputBase_8311D824 :
STRUCT
	{attribute addProperty Name "AdsAddr"}
	AdsAddr AT %I* : AMSADDR;
	{attribute addProperty Name "State"}
	State AT %I* : UINT;
END_STRUCT
END_TYPE

// ---- DUTs/IO/PDOs/Channel_70C997F3.TcDUT
{attribute 'GeneratedUsingTerminal: KL2300-0100'}
{attribute addProperty BoxType "KL2300-0100"}
{attribute addProperty Id "InputAT %I*BOOL0OutputAT %Q*BOOL0"}
{attribute addProperty CRC "1892259827"}
{attribute addProperty Size "0"}
TYPE Channel_70C997F3 :
STRUCT
	{attribute addProperty Name "Input"}
	Input AT %I* : BOOL;
	{attribute addProperty Name "Output"}
	Output AT %Q* : BOOL;
END_STRUCT
END_TYPE

// ---- DUTs/IO/PDOs/EPM_Inputs_Channel_385E794A.TcDUT
{attribute 'GeneratedUsingTerminal: CU2508-0000-0017'}
{attribute addProperty BoxType "CU2508-0000-0017"}
{attribute addProperty Id "Dropped_frames_rxAT %I*USINT1Dropped_frames_txAT %I*USINT1"}
{attribute addProperty CRC "945715530"}
{attribute addProperty Size "2"}
TYPE EPM_Inputs_Channel_385E794A EXTENDS InputBase_8311D824 :
STRUCT
	{attribute addProperty Name "Dropped_frames_rx"}
	Dropped_frames_rx AT %I* : USINT;
	{attribute addProperty Name "Dropped_frames_tx"}
	Dropped_frames_tx AT %I* : USINT;
END_STRUCT
END_TYPE

// ---- DUTs/IO/PDOs/EMPTY_STRUCTURE.TcDUT
{attribute 'GeneratedUsingTerminal: CX5010 EtherCAT slave-1b82-0016'}
{attribute addProperty BoxType "CX5010 EtherCAT slave-1b82-0016"}
{attribute addProperty Id "EMPTY_STRUCTURE"}
{attribute addProperty CRC "0"}
{attribute addProperty Size "0"}
TYPE EMPTY_STRUCTURE :
STRUCT
END_STRUCT
END_TYPE

// ---- DUTs/IO/PDOs/Device_Status_Mapping_61F79077.TcDUT
{attribute 'GeneratedUsingTerminal: CX5010 EtherCAT slave-1b82-0016'}
{attribute addProperty BoxType "CX5010 EtherCAT slave-1b82-0016"}
{attribute addProperty Id "TxPdoStateAT %I*BOOL1TxPdoToggleAT %I*BOOL1"}
{attribute addProperty CRC "1643614327"}
{attribute addProperty Size "2"}
TYPE Device_Status_Mapping_61F79077 EXTENDS InputBase_8311D824 :
STRUCT
	{attribute addProperty Name "TxPdoState"}
	TxPdoState AT %I* : BOOL;
	{attribute addProperty Name "TxPdoToggle"}
	TxPdoToggle AT %I* : BOOL;
END_STRUCT
END_TYPE

// ---- DUTs/IO/PDOs/Channel_954C2EED.TcDUT
{attribute 'GeneratedUsingTerminal: KL9940-0050'}
{attribute addProperty BoxType "KL9940-0050"}
{attribute addProperty Id "Key_1AT %I*BOOL0Key_2AT %I*BOOL0Key_3AT %I*BOOL0Key_4AT %I*BOOL0Key_5AT %I*BOOL0Key_6AT %I*BOOL0Key_7AT %I*BOOL0Key_8AT %I*BOOL0Key_9AT %I*BOOL0Key_10AT %I*BOOL0Key_11AT %I*BOOL0Key_12AT %I*BOOL0Key_13AT %I*BOOL0Key_14AT %I*BOOL0Key_15AT %I*BOOL0Key_16AT %I*BOOL0Key_17AT %I*BOOL0Key_18AT %I*BOOL0Key_19AT %I*BOOL0Key_20AT %I*BOOL0Key_21AT %I*BOOL0Key_22AT %I*BOOL0Key_23AT %I*BOOL0Key_24AT %I*BOOL0Key_25AT %I*BOOL0Key_26AT %I*BOOL0Key_27AT %I*BOOL0Key_28AT %I*BOOL0Key_29AT %I*BOOL0Key_30AT %I*BOOL0Key_31AT %I*BOOL0Key_32AT %I*BOOL0Key_33AT %I*BOOL0Key_34AT %I*BOOL0Key_35AT %I*BOOL0Key_36AT %I*BOOL0Key_37AT %I*BOOL0Key_38AT %I*BOOL0Key_39AT %I*BOOL0Key_40AT %I*BOOL0"}
{attribute addProperty CRC "2504797933"}
{attribute addProperty Size "0"}
TYPE Channel_954C2EED EXTENDS InputBase_8311D824 :
STRUCT
	{attribute addProperty Name "Key_1"}
	Key_1 AT %I* : BOOL;
	{attribute addProperty Name "Key_2"}
	Key_2 AT %I* : BOOL;
	{attribute addProperty Name "Key_3"}
	Key_3 AT %I* : BOOL;
	{attribute addProperty Name "Key_4"}
	Key_4 AT %I* : BOOL;
	{attribute addProperty Name "Key_5"}
	Key_5 AT %I* : BOOL;
	{attribute addProperty Name "Key_6"}
	Key_6 AT %I* : BOOL;
	{attribute addProperty Name "Key_7"}
	Key_7 AT %I* : BOOL;
	{attribute addProperty Name "Key_8"}
	Key_8 AT %I* : BOOL;
	{attribute addProperty Name "Key_9"}
	Key_9 AT %I* : BOOL;
	{attribute addProperty Name "Key_10"}
	Key_10 AT %I* : BOOL;
	{attribute addProperty Name "Key_11"}
	Key_11 AT %I* : BOOL;
	{attribute addProperty Name "Key_12"}
	Key_12 AT %I* : BOOL;
	{attribute addProperty Name "Key_13"}
	Key_13 AT %I* : BOOL;
	{attribute addProperty Name "Key_14"}
	Key_14 AT %I* : BOOL;
	{attribute addProperty Name "Key_15"}
	Key_15 AT %I* : BOOL;
	{attribute addProperty Name "Key_16"}
	Key_16 AT %I* : BOOL;
	{attribute addProperty Name "Key_17"}
	Key_17 AT %I* : BOOL;
	{attribute addProperty Name "Key_18"}
	Key_18 AT %I* : BOOL;
	{attribute addProperty Name "Key_19"}
	Key_19 AT %I* : BOOL;
	{attribute addProperty Name "Key_20"}
	Key_20 AT %I* : BOOL;
	{attribute addProperty Name "Key_21"}
	Key_21 AT %I* : BOOL;
	{attribute addProperty Name "Key_22"}
	Key_22 AT %I* : BOOL;
	{attribute addProperty Name "Key_23"}
	Key_23 AT %I* : BOOL;
	{attribute addProperty Name "Key_24"}
	Key_24 AT %I* : BOOL;
	{attribute addProperty Name "Key_25"}
	Key_25 AT %I* : BOOL;
	{attribute addProperty Name "Key_26"}
	Key_26 AT %I* : BOOL;
	{attribute addProperty Name "Key_27"}
	Key_27 AT %I* : BOOL;
	{attribute addProperty Name "Key_28"}
	Key_28 AT %I* : BOOL;
	{attribute addProperty Name "Key_29"}
	Key_29 AT %I* : BOOL;
	{attribute addProperty Name "Key_30"}
	Key_30 AT %I* : BOOL;
	{attribute addProperty Name "Key_31"}
	Key_31 AT %I* : BOOL;
	{attribute addProperty Name "Key_32"}
	Key_32 AT %I* : BOOL;
	{attribute addProperty Name "Key_33"}
	Key_33 AT %I* : BOOL;
	{attribute addProperty Name "Key_34"}
	Key_34 AT %I* : BOOL;
	{attribute addProperty Name "Key_35"}
	Key_35 AT %I* : BOOL;
	{attribute addProperty Name "Key_36"}
	Key_36 AT %I* : BOOL;
	{attribute addProperty Name "Key_37"}
	Key_37 AT %I* : BOOL;
	{attribute addProperty Name "Key_38"}
	Key_38 AT %I* : BOOL;
	{attribute addProperty Name "Key_39"}
	Key_39 AT %I* : BOOL;
	{attribute addProperty Name "Key_40"}
	Key_40 AT %I* : BOOL;
END_STRUCT
END_TYPE

// ---- DUTs/IO/PDOs/Channel_60E28ED2.TcDUT
{attribute 'GeneratedUsingTerminal: KL9900-0054'}
{attribute addProperty BoxType "KL9900-0054"}
{attribute addProperty Id "Key_1AT %I*BOOL0Key_2AT %I*BOOL0Key_3AT %I*BOOL0Key_4AT %I*BOOL0LED_1AT %Q*BOOL0LED_2AT %Q*BOOL0LED_3AT %Q*BOOL0LED_4AT %Q*BOOL0"}
{attribute addProperty CRC "1625460434"}
{attribute addProperty Size "0"}
TYPE Channel_60E28ED2 :
STRUCT
	{attribute addProperty Name "Key_1"}
	Key_1 AT %I* : BOOL;
	{attribute addProperty Name "Key_2"}
	Key_2 AT %I* : BOOL;
	{attribute addProperty Name "Key_3"}
	Key_3 AT %I* : BOOL;
	{attribute addProperty Name "Key_4"}
	Key_4 AT %I* : BOOL;
	{attribute addProperty Name "LED_1"}
	LED_1 AT %Q* : BOOL;
	{attribute addProperty Name "LED_2"}
	LED_2 AT %Q* : BOOL;
	{attribute addProperty Name "LED_3"}
	LED_3 AT %Q* : BOOL;
	{attribute addProperty Name "LED_4"}
	LED_4 AT %Q* : BOOL;
END_STRUCT
END_TYPE

// ---- DUTs/IO/PDOs/Channel_7DE26195.TcDUT
{attribute 'GeneratedUsingTerminal: KL9900-0055'}
{attribute addProperty BoxType "KL9900-0055"}
{attribute addProperty Id "Key_1AT %I*BOOL0Key_2AT %I*BOOL0Key_3AT %I*BOOL0Key_4AT %I*BOOL0Key_5AT %I*BOOL0Key_6AT %I*BOOL0Key_7AT %I*BOOL0Key_8AT %I*BOOL0LED_1AT %Q*BOOL0LED_2AT %Q*BOOL0LED_3AT %Q*BOOL0LED_4AT %Q*BOOL0LED_5AT %Q*BOOL0LED_6AT %Q*BOOL0LED_7AT %Q*BOOL0LED_8AT %Q*BOOL0"}
{attribute addProperty CRC "2111988117"}
{attribute addProperty Size "0"}
TYPE Channel_7DE26195 :
STRUCT
	{attribute addProperty Name "Key_1"}
	Key_1 AT %I* : BOOL;
	{attribute addProperty Name "Key_2"}
	Key_2 AT %I* : BOOL;
	{attribute addProperty Name "Key_3"}
	Key_3 AT %I* : BOOL;
	{attribute addProperty Name "Key_4"}
	Key_4 AT %I* : BOOL;
	{attribute addProperty Name "Key_5"}
	Key_5 AT %I* : BOOL;
	{attribute addProperty Name "Key_6"}
	Key_6 AT %I* : BOOL;
	{attribute addProperty Name "Key_7"}
	Key_7 AT %I* : BOOL;
	{attribute addProperty Name "Key_8"}
	Key_8 AT %I* : BOOL;
	{attribute addProperty Name "LED_1"}
	LED_1 AT %Q* : BOOL;
	{attribute addProperty Name "LED_2"}
	LED_2 AT %Q* : BOOL;
	{attribute addProperty Name "LED_3"}
	LED_3 AT %Q* : BOOL;
	{attribute addProperty Name "LED_4"}
	LED_4 AT %Q* : BOOL;
	{attribute addProperty Name "LED_5"}
	LED_5 AT %Q* : BOOL;
	{attribute addProperty Name "LED_6"}
	LED_6 AT %Q* : BOOL;
	{attribute addProperty Name "LED_7"}
	LED_7 AT %Q* : BOOL;
	{attribute addProperty Name "LED_8"}
	LED_8 AT %Q* : BOOL;
END_STRUCT
END_TYPE

// ---- DUTs/IO/PDOs/Channel_2E0D480D.TcDUT
{attribute 'GeneratedUsingTerminal: KL9900-0056'}
{attribute addProperty BoxType "KL9900-0056"}
{attribute addProperty Id "Key_1AT %I*BOOL0Key_2AT %I*BOOL0Key_3AT %I*BOOL0Key_4AT %I*BOOL0Key_5AT %I*BOOL0Key_6AT %I*BOOL0Key_7AT %I*BOOL0Key_8AT %I*BOOL0Key_9AT %I*BOOL0Key_10AT %I*BOOL0Key_11AT %I*BOOL0Key_12AT %I*BOOL0LED_1AT %Q*BOOL0LED_2AT %Q*BOOL0LED_3AT %Q*BOOL0LED_4AT %Q*BOOL0LED_5AT %Q*BOOL0LED_6AT %Q*BOOL0LED_7AT %Q*BOOL0LED_8AT %Q*BOOL0LED_9AT %Q*BOOL0LED_10AT %Q*BOOL0LED_11AT %Q*BOOL0LED_12AT %Q*BOOL0"}
{attribute addProperty CRC "772622349"}
{attribute addProperty Size "0"}
TYPE Channel_2E0D480D :
STRUCT
	{attribute addProperty Name "Key_1"}
	Key_1 AT %I* : BOOL;
	{attribute addProperty Name "Key_2"}
	Key_2 AT %I* : BOOL;
	{attribute addProperty Name "Key_3"}
	Key_3 AT %I* : BOOL;
	{attribute addProperty Name "Key_4"}
	Key_4 AT %I* : BOOL;
	{attribute addProperty Name "Key_5"}
	Key_5 AT %I* : BOOL;
	{attribute addProperty Name "Key_6"}
	Key_6 AT %I* : BOOL;
	{attribute addProperty Name "Key_7"}
	Key_7 AT %I* : BOOL;
	{attribute addProperty Name "Key_8"}
	Key_8 AT %I* : BOOL;
	{attribute addProperty Name "Key_9"}
	Key_9 AT %I* : BOOL;
	{attribute addProperty Name "Key_10"}
	Key_10 AT %I* : BOOL;
	{attribute addProperty Name "Key_11"}
	Key_11 AT %I* : BOOL;
	{attribute addProperty Name "Key_12"}
	Key_12 AT %I* : BOOL;
	{attribute addProperty Name "LED_1"}
	LED_1 AT %Q* : BOOL;
	{attribute addProperty Name "LED_2"}
	LED_2 AT %Q* : BOOL;
	{attribute addProperty Name "LED_3"}
	LED_3 AT %Q* : BOOL;
	{attribute addProperty Name "LED_4"}
	LED_4 AT %Q* : BOOL;
	{attribute addProperty Name "LED_5"}
	LED_5 AT %Q* : BOOL;
	{attribute addProperty Name "LED_6"}
	LED_6 AT %Q* : BOOL;
	{attribute addProperty Name "LED_7"}
	LED_7 AT %Q* : BOOL;
	{attribute addProperty Name "LED_8"}
	LED_8 AT %Q* : BOOL;
	{attribute addProperty Name "LED_9"}
	LED_9 AT %Q* : BOOL;
	{attribute addProperty Name "LED_10"}
	LED_10 AT %Q* : BOOL;
	{attribute addProperty Name "LED_11"}
	LED_11 AT %Q* : BOOL;
	{attribute addProperty Name "LED_12"}
	LED_12 AT %Q* : BOOL;
END_STRUCT
END_TYPE

// ---- DUTs/IO/PDOs/Channel_61FC1536.TcDUT
{attribute 'GeneratedUsingTerminal: KL9900-0057'}
{attribute addProperty BoxType "KL9900-0057"}
{attribute addProperty Id "Key_1AT %I*BOOL0Key_2AT %I*BOOL0Key_3AT %I*BOOL0Key_4AT %I*BOOL0Key_5AT %I*BOOL0Key_6AT %I*BOOL0Key_7AT %I*BOOL0Key_8AT %I*BOOL0Key_9AT %I*BOOL0Key_10AT %I*BOOL0Key_11AT %I*BOOL0Key_12AT %I*BOOL0Key_13AT %I*BOOL0Key_14AT %I*BOOL0Key_15AT %I*BOOL0Key_16AT %I*BOOL0LED_1AT %Q*BOOL0LED_2AT %Q*BOOL0LED_3AT %Q*BOOL0LED_4AT %Q*BOOL0LED_5AT %Q*BOOL0LED_6AT %Q*BOOL0LED_7AT %Q*BOOL0LED_8AT %Q*BOOL0LED_9AT %Q*BOOL0LED_10AT %Q*BOOL0LED_11AT %Q*BOOL0LED_12AT %Q*BOOL0LED_13AT %Q*BOOL0LED_14AT %Q*BOOL0LED_15AT %Q*BOOL0LED_16AT %Q*BOOL0"}
{attribute addProperty CRC "1643910454"}
{attribute addProperty Size "0"}
TYPE Channel_61FC1536 :
STRUCT
	{attribute addProperty Name "Key_1"}
	Key_1 AT %I* : BOOL;
	{attribute addProperty Name "Key_2"}
	Key_2 AT %I* : BOOL;
	{attribute addProperty Name "Key_3"}
	Key_3 AT %I* : BOOL;
	{attribute addProperty Name "Key_4"}
	Key_4 AT %I* : BOOL;
	{attribute addProperty Name "Key_5"}
	Key_5 AT %I* : BOOL;
	{attribute addProperty Name "Key_6"}
	Key_6 AT %I* : BOOL;
	{attribute addProperty Name "Key_7"}
	Key_7 AT %I* : BOOL;
	{attribute addProperty Name "Key_8"}
	Key_8 AT %I* : BOOL;
	{attribute addProperty Name "Key_9"}
	Key_9 AT %I* : BOOL;
	{attribute addProperty Name "Key_10"}
	Key_10 AT %I* : BOOL;
	{attribute addProperty Name "Key_11"}
	Key_11 AT %I* : BOOL;
	{attribute addProperty Name "Key_12"}
	Key_12 AT %I* : BOOL;
	{attribute addProperty Name "Key_13"}
	Key_13 AT %I* : BOOL;
	{attribute addProperty Name "Key_14"}
	Key_14 AT %I* : BOOL;
	{attribute addProperty Name "Key_15"}
	Key_15 AT %I* : BOOL;
	{attribute addProperty Name "Key_16"}
	Key_16 AT %I* : BOOL;
	{attribute addProperty Name "LED_1"}
	LED_1 AT %Q* : BOOL;
	{attribute addProperty Name "LED_2"}
	LED_2 AT %Q* : BOOL;
	{attribute addProperty Name "LED_3"}
	LED_3 AT %Q* : BOOL;
	{attribute addProperty Name "LED_4"}
	LED_4 AT %Q* : BOOL;
	{attribute addProperty Name "LED_5"}
	LED_5 AT %Q* : BOOL;
	{attribute addProperty Name "LED_6"}
	LED_6 AT %Q* : BOOL;
	{attribute addProperty Name "LED_7"}
	LED_7 AT %Q* : BOOL;
	{attribute addProperty Name "LED_8"}
	LED_8 AT %Q* : BOOL;
	{attribute addProperty Name "LED_9"}
	LED_9 AT %Q* : BOOL;
	{attribute addProperty Name "LED_10"}
	LED_10 AT %Q* : BOOL;
	{attribute addProperty Name "LED_11"}
	LED_11 AT %Q* : BOOL;
	{attribute addProperty Name "LED_12"}
	LED_12 AT %Q* : BOOL;
	{attribute addProperty Name "LED_13"}
	LED_13 AT %Q* : BOOL;
	{attribute addProperty Name "LED_14"}
	LED_14 AT %Q* : BOOL;
	{attribute addProperty Name "LED_15"}
	LED_15 AT %Q* : BOOL;
	{attribute addProperty Name "LED_16"}
	LED_16 AT %Q* : BOOL;
END_STRUCT
END_TYPE

// ---- DUTs/IO/PDOs/Channel_16463F74.TcDUT
{attribute 'GeneratedUsingTerminal: KL9900-0058'}
{attribute addProperty BoxType "KL9900-0058"}
{attribute addProperty Id "Key_1AT %I*BOOL0Key_2AT %I*BOOL0Key_3AT %I*BOOL0Key_4AT %I*BOOL0Key_5AT %I*BOOL0Key_6AT %I*BOOL0Key_7AT %I*BOOL0Key_8AT %I*BOOL0Key_9AT %I*BOOL0Key_10AT %I*BOOL0Key_11AT %I*BOOL0Key_12AT %I*BOOL0Key_13AT %I*BOOL0Key_14AT %I*BOOL0Key_15AT %I*BOOL0Key_16AT %I*BOOL0Key_17AT %I*BOOL0Key_18AT %I*BOOL0Key_19AT %I*BOOL0Key_20AT %I*BOOL0LED_1AT %Q*BOOL0LED_2AT %Q*BOOL0LED_3AT %Q*BOOL0LED_4AT %Q*BOOL0LED_5AT %Q*BOOL0LED_6AT %Q*BOOL0LED_7AT %Q*BOOL0LED_8AT %Q*BOOL0LED_9AT %Q*BOOL0LED_10AT %Q*BOOL0LED_11AT %Q*BOOL0LED_12AT %Q*BOOL0LED_13AT %Q*BOOL0LED_14AT %Q*BOOL0LED_15AT %Q*BOOL0LED_16AT %Q*BOOL0LED_17AT %Q*BOOL0LED_18AT %Q*BOOL0LED_19AT %Q*BOOL0LED_20AT %Q*BOOL0"}
{attribute addProperty CRC "373702516"}
{attribute addProperty Size "0"}
TYPE Channel_16463F74 :
STRUCT
	{attribute addProperty Name "Key_1"}
	Key_1 AT %I* : BOOL;
	{attribute addProperty Name "Key_2"}
	Key_2 AT %I* : BOOL;
	{attribute addProperty Name "Key_3"}
	Key_3 AT %I* : BOOL;
	{attribute addProperty Name "Key_4"}
	Key_4 AT %I* : BOOL;
	{attribute addProperty Name "Key_5"}
	Key_5 AT %I* : BOOL;
	{attribute addProperty Name "Key_6"}
	Key_6 AT %I* : BOOL;
	{attribute addProperty Name "Key_7"}
	Key_7 AT %I* : BOOL;
	{attribute addProperty Name "Key_8"}
	Key_8 AT %I* : BOOL;
	{attribute addProperty Name "Key_9"}
	Key_9 AT %I* : BOOL;
	{attribute addProperty Name "Key_10"}
	Key_10 AT %I* : BOOL;
	{attribute addProperty Name "Key_11"}
	Key_11 AT %I* : BOOL;
	{attribute addProperty Name "Key_12"}
	Key_12 AT %I* : BOOL;
	{attribute addProperty Name "Key_13"}
	Key_13 AT %I* : BOOL;
	{attribute addProperty Name "Key_14"}
	Key_14 AT %I* : BOOL;
	{attribute addProperty Name "Key_15"}
	Key_15 AT %I* : BOOL;
	{attribute addProperty Name "Key_16"}
	Key_16 AT %I* : BOOL;
	{attribute addProperty Name "Key_17"}
	Key_17 AT %I* : BOOL;
	{attribute addProperty Name "Key_18"}
	Key_18 AT %I* : BOOL;
	{attribute addProperty Name "Key_19"}
	Key_19 AT %I* : BOOL;
	{attribute addProperty Name "Key_20"}
	Key_20 AT %I* : BOOL;
	{attribute addProperty Name "LED_1"}
	LED_1 AT %Q* : BOOL;
	{attribute addProperty Name "LED_2"}
	LED_2 AT %Q* : BOOL;
	{attribute addProperty Name "LED_3"}
	LED_3 AT %Q* : BOOL;
	{attribute addProperty Name "LED_4"}
	LED_4 AT %Q* : BOOL;
	{attribute addProperty Name "LED_5"}
	LED_5 AT %Q* : BOOL;
	{attribute addProperty Name "LED_6"}
	LED_6 AT %Q* : BOOL;
	{attribute addProperty Name "LED_7"}
	LED_7 AT %Q* : BOOL;
	{attribute addProperty Name "LED_8"}
	LED_8 AT %Q* : BOOL;
	{attribute addProperty Name "LED_9"}
	LED_9 AT %Q* : BOOL;
	{attribute addProperty Name "LED_10"}
	LED_10 AT %Q* : BOOL;
	{attribute addProperty Name "LED_11"}
	LED_11 AT %Q* : BOOL;
	{attribute addProperty Name "LED_12"}
	LED_12 AT %Q* : BOOL;
	{attribute addProperty Name "LED_13"}
	LED_13 AT %Q* : BOOL;
	{attribute addProperty Name "LED_14"}
	LED_14 AT %Q* : BOOL;
	{attribute addProperty Name "LED_15"}
	LED_15 AT %Q* : BOOL;
	{attribute addProperty Name "LED_16"}
	LED_16 AT %Q* : BOOL;
	{attribute addProperty Name "LED_17"}
	LED_17 AT %Q* : BOOL;
	{attribute addProperty Name "LED_18"}
	LED_18 AT %Q* : BOOL;
	{attribute addProperty Name "LED_19"}
	LED_19 AT %Q* : BOOL;
	{attribute addProperty Name "LED_20"}
	LED_20 AT %Q* : BOOL;
END_STRUCT
END_TYPE

// ---- DUTs/IO/PDOs/Channel_707BD1FE.TcDUT
{attribute 'GeneratedUsingTerminal: KL9900-0059'}
{attribute addProperty BoxType "KL9900-0059"}
{attribute addProperty Id "Key_1AT %I*BOOL0Key_2AT %I*BOOL0Key_3AT %I*BOOL0Key_4AT %I*BOOL0Key_5AT %I*BOOL0Key_6AT %I*BOOL0Key_7AT %I*BOOL0Key_8AT %I*BOOL0Key_9AT %I*BOOL0Key_10AT %I*BOOL0Key_11AT %I*BOOL0Key_12AT %I*BOOL0Key_13AT %I*BOOL0Key_14AT %I*BOOL0Key_15AT %I*BOOL0Key_16AT %I*BOOL0Key_17AT %I*BOOL0Key_18AT %I*BOOL0Key_19AT %I*BOOL0Key_20AT %I*BOOL0Key_21AT %I*BOOL0Key_22AT %I*BOOL0Key_23AT %I*BOOL0Key_24AT %I*BOOL0LED_1AT %Q*BOOL0LED_2AT %Q*BOOL0LED_3AT %Q*BOOL0LED_4AT %Q*BOOL0LED_5AT %Q*BOOL0LED_6AT %Q*BOOL0LED_7AT %Q*BOOL0LED_8AT %Q*BOOL0LED_9AT %Q*BOOL0LED_10AT %Q*BOOL0LED_11AT %Q*BOOL0LED_12AT %Q*BOOL0LED_13AT %Q*BOOL0LED_14AT %Q*BOOL0LED_15AT %Q*BOOL0LED_16AT %Q*BOOL0LED_17AT %Q*BOOL0LED_18AT %Q*BOOL0LED_19AT %Q*BOOL0LED_20AT %Q*BOOL0LED_21AT %Q*BOOL0LED_22AT %Q*BOOL0LED_23AT %Q*BOOL0LED_24AT %Q*BOOL0"}
{attribute addProperty CRC "1887162878"}
{attribute addProperty Size "0"}
TYPE Channel_707BD1FE :
STRUCT
	{attribute addProperty Name "Key_1"}
	Key_1 AT %I* : BOOL;
	{attribute addProperty Name "Key_2"}
	Key_2 AT %I* : BOOL;
	{attribute addProperty Name "Key_3"}
	Key_3 AT %I* : BOOL;
	{attribute addProperty Name "Key_4"}
	Key_4 AT %I* : BOOL;
	{attribute addProperty Name "Key_5"}
	Key_5 AT %I* : BOOL;
	{attribute addProperty Name "Key_6"}
	Key_6 AT %I* : BOOL;
	{attribute addProperty Name "Key_7"}
	Key_7 AT %I* : BOOL;
	{attribute addProperty Name "Key_8"}
	Key_8 AT %I* : BOOL;
	{attribute addProperty Name "Key_9"}
	Key_9 AT %I* : BOOL;
	{attribute addProperty Name "Key_10"}
	Key_10 AT %I* : BOOL;
	{attribute addProperty Name "Key_11"}
	Key_11 AT %I* : BOOL;
	{attribute addProperty Name "Key_12"}
	Key_12 AT %I* : BOOL;
	{attribute addProperty Name "Key_13"}
	Key_13 AT %I* : BOOL;
	{attribute addProperty Name "Key_14"}
	Key_14 AT %I* : BOOL;
	{attribute addProperty Name "Key_15"}
	Key_15 AT %I* : BOOL;
	{attribute addProperty Name "Key_16"}
	Key_16 AT %I* : BOOL;
	{attribute addProperty Name "Key_17"}
	Key_17 AT %I* : BOOL;
	{attribute addProperty Name "Key_18"}
	Key_18 AT %I* : BOOL;
	{attribute addProperty Name "Key_19"}
	Key_19 AT %I* : BOOL;
	{attribute addProperty Name "Key_20"}
	Key_20 AT %I* : BOOL;
	{attribute addProperty Name "Key_21"}
	Key_21 AT %I* : BOOL;
	{attribute addProperty Name "Key_22"}
	Key_22 AT %I* : BOOL;
	{attribute addProperty Name "Key_23"}
	Key_23 AT %I* : BOOL;
	{attribute addProperty Name "Key_24"}
	Key_24 AT %I* : BOOL;
	{attribute addProperty Name "LED_1"}
	LED_1 AT %Q* : BOOL;
	{attribute addProperty Name "LED_2"}
	LED_2 AT %Q* : BOOL;
	{attribute addProperty Name "LED_3"}
	LED_3 AT %Q* : BOOL;
	{attribute addProperty Name "LED_4"}
	LED_4 AT %Q* : BOOL;
	{attribute addProperty Name "LED_5"}
	LED_5 AT %Q* : BOOL;
	{attribute addProperty Name "LED_6"}
	LED_6 AT %Q* : BOOL;
	{attribute addProperty Name "LED_7"}
	LED_7 AT %Q* : BOOL;
	{attribute addProperty Name "LED_8"}
	LED_8 AT %Q* : BOOL;
	{attribute addProperty Name "LED_9"}
	LED_9 AT %Q* : BOOL;
	{attribute addProperty Name "LED_10"}
	LED_10 AT %Q* : BOOL;
	{attribute addProperty Name "LED_11"}
	LED_11 AT %Q* : BOOL;
	{attribute addProperty Name "LED_12"}
	LED_12 AT %Q* : BOOL;
	{attribute addProperty Name "LED_13"}
	LED_13 AT %Q* : BOOL;
	{attribute addProperty Name "LED_14"}
	LED_14 AT %Q* : BOOL;
	{attribute addProperty Name "LED_15"}
	LED_15 AT %Q* : BOOL;
	{attribute addProperty Name "LED_16"}
	LED_16 AT %Q* : BOOL;
	{attribute addProperty Name "LED_17"}
	LED_17 AT %Q* : BOOL;
	{attribute addProperty Name "LED_18"}
	LED_18 AT %Q* : BOOL;
	{attribute addProperty Name "LED_19"}
	LED_19 AT %Q* : BOOL;
	{attribute addProperty Name "LED_20"}
	LED_20 AT %Q* : BOOL;
	{attribute addProperty Name "LED_21"}
	LED_21 AT %Q* : BOOL;
	{attribute addProperty Name "LED_22"}
	LED_22 AT %Q* : BOOL;
	{attribute addProperty Name "LED_23"}
	LED_23 AT %Q* : BOOL;
	{attribute addProperty Name "LED_24"}
	LED_24 AT %Q* : BOOL;
END_STRUCT
END_TYPE

// ---- DUTs/IO/PDOs/Channel_7D202F58.TcDUT
{attribute 'GeneratedUsingTerminal: KL9900-0060'}
{attribute addProperty BoxType "KL9900-0060"}
{attribute addProperty Id "Key_1AT %I*BOOL0Key_2AT %I*BOOL0Key_3AT %I*BOOL0Key_4AT %I*BOOL0Key_5AT %I*BOOL0Key_6AT %I*BOOL0Key_7AT %I*BOOL0Key_8AT %I*BOOL0Key_9AT %I*BOOL0Key_10AT %I*BOOL0Key_11AT %I*BOOL0Key_12AT %I*BOOL0Key_13AT %I*BOOL0Key_14AT %I*BOOL0Key_15AT %I*BOOL0Key_16AT %I*BOOL0Key_17AT %I*BOOL0Key_18AT %I*BOOL0Key_19AT %I*BOOL0Key_20AT %I*BOOL0Key_21AT %I*BOOL0Key_22AT %I*BOOL0Key_23AT %I*BOOL0Key_24AT %I*BOOL0Key_25AT %I*BOOL0Key_26AT %I*BOOL0Key_27AT %I*BOOL0Key_28AT %I*BOOL0LED_1AT %Q*BOOL0LED_2AT %Q*BOOL0LED_3AT %Q*BOOL0LED_4AT %Q*BOOL0LED_5AT %Q*BOOL0LED_6AT %Q*BOOL0LED_7AT %Q*BOOL0LED_8AT %Q*BOOL0LED_9AT %Q*BOOL0LED_10AT %Q*BOOL0LED_11AT %Q*BOOL0LED_12AT %Q*BOOL0LED_13AT %Q*BOOL0LED_14AT %Q*BOOL0LED_15AT %Q*BOOL0LED_16AT %Q*BOOL0LED_17AT %Q*BOOL0LED_18AT %Q*BOOL0LED_19AT %Q*BOOL0LED_20AT %Q*BOOL0LED_21AT %Q*BOOL0LED_22AT %Q*BOOL0LED_23AT %Q*BOOL0LED_24AT %Q*BOOL0LED_25AT %Q*BOOL0LED_26AT %Q*BOOL0LED_27AT %Q*BOOL0LED_28AT %Q*BOOL0"}
{attribute addProperty CRC "2099261272"}
{attribute addProperty Size "0"}
TYPE Channel_7D202F58 :
STRUCT
	{attribute addProperty Name "Key_1"}
	Key_1 AT %I* : BOOL;
	{attribute addProperty Name "Key_2"}
	Key_2 AT %I* : BOOL;
	{attribute addProperty Name "Key_3"}
	Key_3 AT %I* : BOOL;
	{attribute addProperty Name "Key_4"}
	Key_4 AT %I* : BOOL;
	{attribute addProperty Name "Key_5"}
	Key_5 AT %I* : BOOL;
	{attribute addProperty Name "Key_6"}
	Key_6 AT %I* : BOOL;
	{attribute addProperty Name "Key_7"}
	Key_7 AT %I* : BOOL;
	{attribute addProperty Name "Key_8"}
	Key_8 AT %I* : BOOL;
	{attribute addProperty Name "Key_9"}
	Key_9 AT %I* : BOOL;
	{attribute addProperty Name "Key_10"}
	Key_10 AT %I* : BOOL;
	{attribute addProperty Name "Key_11"}
	Key_11 AT %I* : BOOL;
	{attribute addProperty Name "Key_12"}
	Key_12 AT %I* : BOOL;
	{attribute addProperty Name "Key_13"}
	Key_13 AT %I* : BOOL;
	{attribute addProperty Name "Key_14"}
	Key_14 AT %I* : BOOL;
	{attribute addProperty Name "Key_15"}
	Key_15 AT %I* : BOOL;
	{attribute addProperty Name "Key_16"}
	Key_16 AT %I* : BOOL;
	{attribute addProperty Name "Key_17"}
	Key_17 AT %I* : BOOL;
	{attribute addProperty Name "Key_18"}
	Key_18 AT %I* : BOOL;
	{attribute addProperty Name "Key_19"}
	Key_19 AT %I* : BOOL;
	{attribute addProperty Name "Key_20"}
	Key_20 AT %I* : BOOL;
	{attribute addProperty Name "Key_21"}
	Key_21 AT %I* : BOOL;
	{attribute addProperty Name "Key_22"}
	Key_22 AT %I* : BOOL;
	{attribute addProperty Name "Key_23"}
	Key_23 AT %I* : BOOL;
	{attribute addProperty Name "Key_24"}
	Key_24 AT %I* : BOOL;
	{attribute addProperty Name "Key_25"}
	Key_25 AT %I* : BOOL;
	{attribute addProperty Name "Key_26"}
	Key_26 AT %I* : BOOL;
	{attribute addProperty Name "Key_27"}
	Key_27 AT %I* : BOOL;
	{attribute addProperty Name "Key_28"}
	Key_28 AT %I* : BOOL;
	{attribute addProperty Name "LED_1"}
	LED_1 AT %Q* : BOOL;
	{attribute addProperty Name "LED_2"}
	LED_2 AT %Q* : BOOL;
	{attribute addProperty Name "LED_3"}
	LED_3 AT %Q* : BOOL;
	{attribute addProperty Name "LED_4"}
	LED_4 AT %Q* : BOOL;
	{attribute addProperty Name "LED_5"}
	LED_5 AT %Q* : BOOL;
	{attribute addProperty Name "LED_6"}
	LED_6 AT %Q* : BOOL;
	{attribute addProperty Name "LED_7"}
	LED_7 AT %Q* : BOOL;
	{attribute addProperty Name "LED_8"}
	LED_8 AT %Q* : BOOL;
	{attribute addProperty Name "LED_9"}
	LED_9 AT %Q* : BOOL;
	{attribute addProperty Name "LED_10"}
	LED_10 AT %Q* : BOOL;
	{attribute addProperty Name "LED_11"}
	LED_11 AT %Q* : BOOL;
	{attribute addProperty Name "LED_12"}
	LED_12 AT %Q* : BOOL;
	{attribute addProperty Name "LED_13"}
	LED_13 AT %Q* : BOOL;
	{attribute addProperty Name "LED_14"}
	LED_14 AT %Q* : BOOL;
	{attribute addProperty Name "LED_15"}
	LED_15 AT %Q* : BOOL;
	{attribute addProperty Name "LED_16"}
	LED_16 AT %Q* : BOOL;
	{attribute addProperty Name "LED_17"}
	LED_17 AT %Q* : BOOL;
	{attribute addProperty Name "LED_18"}
	LED_18 AT %Q* : BOOL;
	{attribute addProperty Name "LED_19"}
	LED_19 AT %Q* : BOOL;
	{attribute addProperty Name "LED_20"}
	LED_20 AT %Q* : BOOL;
	{attribute addProperty Name "LED_21"}
	LED_21 AT %Q* : BOOL;
	{attribute addProperty Name "LED_22"}
	LED_22 AT %Q* : BOOL;
	{attribute addProperty Name "LED_23"}
	LED_23 AT %Q* : BOOL;
	{attribute addProperty Name "LED_24"}
	LED_24 AT %Q* : BOOL;
	{attribute addProperty Name "LED_25"}
	LED_25 AT %Q* : BOOL;
	{attribute addProperty Name "LED_26"}
	LED_26 AT %Q* : BOOL;
	{attribute addProperty Name "LED_27"}
	LED_27 AT %Q* : BOOL;
	{attribute addProperty Name "LED_28"}
	LED_28 AT %Q* : BOOL;
END_STRUCT
END_TYPE

// ---- DUTs/IO/PDOs/Channel_6CC0E226.TcDUT
{attribute 'GeneratedUsingTerminal: KL9900-0063'}
{attribute addProperty BoxType "KL9900-0063"}
{attribute addProperty Id "Key_1AT %I*BOOL0Key_2AT %I*BOOL0Key_3AT %I*BOOL0Input_1AT %I*BOOL0Input_2AT %I*BOOL0Input_3AT %I*BOOL0LED_1AT %Q*BOOL0LED_2AT %Q*BOOL0LED_3AT %Q*BOOL0"}
{attribute addProperty CRC "1824580134"}
{attribute addProperty Size "0"}
TYPE Channel_6CC0E226 :
STRUCT
	{attribute addProperty Name "Key_1"}
	Key_1 AT %I* : BOOL;
	{attribute addProperty Name "Key_2"}
	Key_2 AT %I* : BOOL;
	{attribute addProperty Name "Key_3"}
	Key_3 AT %I* : BOOL;
	{attribute addProperty Name "Input_1"}
	Input_1 AT %I* : BOOL;
	{attribute addProperty Name "Input_2"}
	Input_2 AT %I* : BOOL;
	{attribute addProperty Name "Input_3"}
	Input_3 AT %I* : BOOL;
	{attribute addProperty Name "LED_1"}
	LED_1 AT %Q* : BOOL;
	{attribute addProperty Name "LED_2"}
	LED_2 AT %Q* : BOOL;
	{attribute addProperty Name "LED_3"}
	LED_3 AT %Q* : BOOL;
END_STRUCT
END_TYPE

// ---- DUTs/IO/PDOs/Channel_0F0CD940.TcDUT
{attribute 'GeneratedUsingTerminal: KL9900-0064'}
{attribute addProperty BoxType "KL9900-0064"}
{attribute addProperty Id "Key_1AT %I*BOOL0Key_2AT %I*BOOL0Key_3AT %I*BOOL0Key_4AT %I*BOOL0Input_1AT %I*BOOL0Input_2AT %I*BOOL0Input_3AT %I*BOOL0Input_4AT %I*BOOL0LED_1AT %Q*BOOL0LED_2AT %Q*BOOL0LED_3AT %Q*BOOL0LED_4AT %Q*BOOL0"}
{attribute addProperty CRC "252500288"}
{attribute addProperty Size "0"}
TYPE Channel_0F0CD940 :
STRUCT
	{attribute addProperty Name "Key_1"}
	Key_1 AT %I* : BOOL;
	{attribute addProperty Name "Key_2"}
	Key_2 AT %I* : BOOL;
	{attribute addProperty Name "Key_3"}
	Key_3 AT %I* : BOOL;
	{attribute addProperty Name "Key_4"}
	Key_4 AT %I* : BOOL;
	{attribute addProperty Name "Input_1"}
	Input_1 AT %I* : BOOL;
	{attribute addProperty Name "Input_2"}
	Input_2 AT %I* : BOOL;
	{attribute addProperty Name "Input_3"}
	Input_3 AT %I* : BOOL;
	{attribute addProperty Name "Input_4"}
	Input_4 AT %I* : BOOL;
	{attribute addProperty Name "LED_1"}
	LED_1 AT %Q* : BOOL;
	{attribute addProperty Name "LED_2"}
	LED_2 AT %Q* : BOOL;
	{attribute addProperty Name "LED_3"}
	LED_3 AT %Q* : BOOL;
	{attribute addProperty Name "LED_4"}
	LED_4 AT %Q* : BOOL;
END_STRUCT
END_TYPE

// ---- DUTs/IO/PDOs/Channel_65B76600.TcDUT
{attribute 'GeneratedUsingTerminal: KL9900-0062'}
{attribute addProperty BoxType "KL9900-0062"}
{attribute addProperty Id "E_StopAT %I*BOOL0"}
{attribute addProperty CRC "1706518016"}
{attribute addProperty Size "0"}
TYPE Channel_65B76600 EXTENDS InputBase_8311D824 :
STRUCT
	{attribute addProperty Name "E_Stop"}
	E_Stop AT %I* : BOOL;
END_STRUCT
END_TYPE

// ---- DUTs/IO/PDOs/Channel_72DF6336.TcDUT
{attribute 'GeneratedUsingTerminal: KL1212'}
{attribute addProperty BoxType "KL1212"}
{attribute addProperty Id "InputAT %I*BOOL0ErrorAT %I*BOOL0PowerAT %Q*BOOL0"}
{attribute addProperty CRC "1927242550"}
{attribute addProperty Size "0"}
TYPE Channel_72DF6336 :
STRUCT
	{attribute addProperty Name "Input"}
	Input AT %I* : BOOL;
	{attribute addProperty Name "Error"}
	Error AT %I* : BOOL;
	{attribute addProperty Name "Power"}
	Power AT %Q* : BOOL;
END_STRUCT
END_TYPE

// ---- DUTs/IO/PDOs/Channel_22DCD695.TcDUT
{attribute 'GeneratedUsingTerminal: KL1352'}
{attribute addProperty BoxType "KL1352"}
{attribute addProperty Id "InputAT %I*BOOL0ErrorAT %I*BOOL0"}
{attribute addProperty CRC "584898197"}
{attribute addProperty Size "0"}
TYPE Channel_22DCD695 EXTENDS InputBase_8311D824 :
STRUCT
	{attribute addProperty Name "Input"}
	Input AT %I* : BOOL;
	{attribute addProperty Name "Error"}
	Error AT %I* : BOOL;
END_STRUCT
END_TYPE

// ---- DUTs/IO/PDOs/Channel_3C1A6500.TcDUT
{attribute 'GeneratedUsingTerminal: KL1501'}
{attribute addProperty BoxType "KL1501"}
{attribute addProperty Id "StateAT %I*USINT0Data_InAT %I*ARRAY [0..1] OF UINT0CtrlAT %Q*USINT0Data_OutAT %Q*ARRAY [0..1] OF UINT0"}
{attribute addProperty CRC "1008362752"}
{attribute addProperty Size "0"}
TYPE Channel_3C1A6500 :
STRUCT
	{attribute addProperty Name "State"}
	State AT %I* : USINT;
	{attribute addProperty Name "Data_In"}
	Data_In AT %I* : ARRAY [0..1] OF UINT;
	{attribute addProperty Name "Ctrl"}
	Ctrl AT %Q* : USINT;
	{attribute addProperty Name "Data_Out"}
	Data_Out AT %Q* : ARRAY [0..1] OF UINT;
END_STRUCT
END_TYPE

// ---- DUTs/IO/PDOs/Channel_B5275D8E.TcDUT
{attribute 'GeneratedUsingTerminal: KL1501-0001'}
{attribute addProperty BoxType "KL1501-0001"}
{attribute addProperty Id "StatusAT %I*USINT0CounterAT %I*UINT0Latch_PeriodLAT %I*UINT0PeriodHAT %I*USINT0CtrlAT %Q*USINT0RegDataAT %Q*UINT0"}
{attribute addProperty CRC "3039255950"}
{attribute addProperty Size "0"}
TYPE Channel_B5275D8E :
STRUCT
	{attribute addProperty Name "Status"}
	Status AT %I* : USINT;
	{attribute addProperty Name "Counter"}
	Counter AT %I* : UINT;
	{attribute addProperty Name "Latch_PeriodL"}
	Latch_PeriodL AT %I* : UINT;
	{attribute addProperty Name "PeriodH"}
	PeriodH AT %I* : USINT;
	{attribute addProperty Name "Ctrl"}
	Ctrl AT %Q* : USINT;
	{attribute addProperty Name "RegData"}
	RegData AT %Q* : UINT;
END_STRUCT
END_TYPE

// ---- DUTs/IO/PDOs/Channel_03CEAA5E.TcDUT
{attribute 'GeneratedUsingTerminal: KL1512'}
{attribute addProperty BoxType "KL1512"}
{attribute addProperty Id "StateAT %I*USINT0Data_InAT %I*UINT0CtrlAT %Q*USINT0Data_OutAT %Q*UINT0"}
{attribute addProperty CRC "63875678"}
{attribute addProperty Size "0"}
TYPE Channel_03CEAA5E :
STRUCT
	{attribute addProperty Name "State"}
	State AT %I* : USINT;
	{attribute addProperty Name "Data_In"}
	Data_In AT %I* : UINT;
	{attribute addProperty Name "Ctrl"}
	Ctrl AT %Q* : USINT;
	{attribute addProperty Name "Data_Out"}
	Data_Out AT %Q* : UINT;
END_STRUCT
END_TYPE

// ---- DUTs/IO/PDOs/Channel_1D6668A9.TcDUT
{attribute 'GeneratedUsingTerminal: KL1904'}
{attribute addProperty BoxType "KL1904"}
{attribute addProperty Id "Safety_InAT %I*ARRAY[0..5] OF BYTE0Safety_OutAT %Q*ARRAY[0..5] OF BYTE0"}
{attribute addProperty CRC "493250729"}
{attribute addProperty Size "0"}
TYPE Channel_1D6668A9 :
STRUCT
	{attribute addProperty Name "Safety_In"}
	Safety_In AT %I* : ARRAY[0..5] OF BYTE;
	{attribute addProperty Name "Safety_Out"}
	Safety_Out AT %Q* : ARRAY[0..5] OF BYTE;
END_STRUCT
END_TYPE

// ---- DUTs/IO/PDOs/Channel_6B723A16.TcDUT
{attribute 'GeneratedUsingTerminal: KL1644-0050'}
{attribute addProperty BoxType "KL1644-0050"}
{attribute addProperty Id "SwitchAT %I*BOOL0OutputAT %Q*BOOL0"}
{attribute addProperty CRC "1802648086"}
{attribute addProperty Size "0"}
TYPE Channel_6B723A16 :
STRUCT
	{attribute addProperty Name "Switch"}
	Switch AT %I* : BOOL;
	{attribute addProperty Name "Output"}
	Output AT %Q* : BOOL;
END_STRUCT
END_TYPE

// ---- DUTs/IO/PDOs/Channel_460B8C40.TcDUT
{attribute 'GeneratedUsingTerminal: KL2012'}
{attribute addProperty BoxType "KL2012"}
{attribute addProperty Id "OutputAT %Q*BOOL0"}
{attribute addProperty CRC "1175161920"}
{attribute addProperty Size "0"}
TYPE Channel_460B8C40 EXTENDS OutputBase_10CEE7DE :
STRUCT
	{attribute addProperty Name "Output"}
	Output AT %Q* : BOOL;
END_STRUCT
END_TYPE

// ---- DUTs/IO/PDOs/Channel_DCF170BB.TcDUT
{attribute 'GeneratedUsingTerminal: KL2212'}
{attribute addProperty BoxType "KL2212"}
{attribute addProperty Id "WireBreakAT %I*BOOL0CurcuitAT %I*BOOL0OutputAT %Q*BOOL0"}
{attribute addProperty CRC "3706810555"}
{attribute addProperty Size "0"}
TYPE Channel_DCF170BB :
STRUCT
	{attribute addProperty Name "WireBreak"}
	WireBreak AT %I* : BOOL;
	{attribute addProperty Name "Curcuit"}
	Curcuit AT %I* : BOOL;
	{attribute addProperty Name "Output"}
	Output AT %Q* : BOOL;
END_STRUCT
END_TYPE

// ---- DUTs/IO/PDOs/Channel_26FC8FD8.TcDUT
{attribute 'GeneratedUsingTerminal: KL2284'}
{attribute addProperty BoxType "KL2284"}
{attribute addProperty Id "CWAT %Q*BOOL0CCWAT %Q*BOOL0"}
{attribute addProperty CRC "654086104"}
{attribute addProperty Size "0"}
TYPE Channel_26FC8FD8 EXTENDS OutputBase_10CEE7DE :
STRUCT
	{attribute addProperty Name "CW"}
	CW AT %Q* : BOOL;
	{attribute addProperty Name "CCW"}
	CCW AT %Q* : BOOL;
END_STRUCT
END_TYPE

// ---- DUTs/IO/PDOs/Channel_FEA3DBF8.TcDUT
{attribute 'GeneratedUsingTerminal: KL2531'}
{attribute addProperty BoxType "KL2531"}
{attribute addProperty Id "StatusAT %I*USINT0PositionAT %I*UINT0ExtStatusAT %I*UINT0CtrlAT %Q*USINT0VelocityAT %Q*INT0ExtCtrlAT %Q*UINT0"}
{attribute addProperty CRC "4272151544"}
{attribute addProperty Size "0"}
TYPE Channel_FEA3DBF8 :
STRUCT
	{attribute addProperty Name "Status"}
	Status AT %I* : USINT;
	{attribute addProperty Name "Position"}
	Position AT %I* : UINT;
	{attribute addProperty Name "ExtStatus"}
	ExtStatus AT %I* : UINT;
	{attribute addProperty Name "Ctrl"}
	Ctrl AT %Q* : USINT;
	{attribute addProperty Name "Velocity"}
	Velocity AT %Q* : INT;
	{attribute addProperty Name "ExtCtrl"}
	ExtCtrl AT %Q* : UINT;
END_STRUCT
END_TYPE

// ---- DUTs/IO/PDOs/Channel_0D1929F0.TcDUT
{attribute 'GeneratedUsingTerminal: KL2531-0001'}
{attribute addProperty BoxType "KL2531-0001"}
{attribute addProperty Id "StatusAT %I*USINT0PositionAT %I*UDINT0ExtStatusAT %I*UINT0CtrlAT %Q*USINT0VelocityAT %Q*DINT0ExtCtrlAT %Q*UINT0"}
{attribute addProperty CRC "219752944"}
{attribute addProperty Size "0"}
TYPE Channel_0D1929F0 :
STRUCT
	{attribute addProperty Name "Status"}
	Status AT %I* : USINT;
	{attribute addProperty Name "Position"}
	Position AT %I* : UDINT;
	{attribute addProperty Name "ExtStatus"}
	ExtStatus AT %I* : UINT;
	{attribute addProperty Name "Ctrl"}
	Ctrl AT %Q* : USINT;
	{attribute addProperty Name "Velocity"}
	Velocity AT %Q* : DINT;
	{attribute addProperty Name "ExtCtrl"}
	ExtCtrl AT %Q* : UINT;
END_STRUCT
END_TYPE

